LIN {X 0,Y 262.502,Z 609.726,A -85,B 0,C 180,E1 11906.298,E2 11906.298} C_VEL
LIN {X 0,Y 258.219,Z 619.545,A -85,B 0,C 180,E1 11905.702,E2 11905.702} C_VEL
LIN {X 0,Y 254.32,Z 626.854,A -85,B 0,C 180,E1 11904.847,E2 11904.847} C_VEL
LIN {X 0,Y 252.122,Z 630.311,A -85,B 0,C 180,E1 11904.198,E2 11904.198} C_VEL
LIN {X 0,Y 248.406,Z 637.947,A -85,B 0,C 180,E1 11903.61,E2 11903.61} C_VEL
LIN {X 0,Y 245.083,Z 643.553,A -85,B 0,C 180,E1 11902.804,E2 11902.804} C_VEL
LIN {X 0,Y 242.242,Z 647.159,A -85,B 0,C 180,E1 11901.808,E2 11901.808} C_VEL
LIN {X 0,Y 241.54,Z 648.252,A -85,B 0,C 180,E1 11901.619,E2 11901.619} C_VEL
LIN {X 0,Y 238.221,Z 654.054,A -85,B 0,C 180,E1 11900.902,E2 11900.902} C_VEL
LIN {X 0,Y 235.659,Z 657.613,A -85,B 0,C 180,E1 11900.102,E2 11900.102} C_VEL
LIN {X 0,Y 234.291,Z 659.07,A -85,B 0,C 180,E1 11899.444,E2 11899.444} C_VEL
LIN {X 0,Y 233.714,Z 659.362,A -85,B 0,C 180,E1 11898.975,E2 11898.975} C_VEL
LIN {X 0,Y 232.454,Z 676.024,A -85,B 0,C 180,E1 11897.008,E2 11897.008} C_VEL
LIN {X 0,Y 231.033,Z 692.343,A -85,B 0,C 180,E1 11894.538,E2 11894.538} C_VEL
LIN {X 0,Y 229.738,Z 706.728,A -85,B 0,C 180,E1 11891.804,E2 11891.804} C_VEL
LIN {X 0,Y 228.67,Z 719.328,A -85,B 0,C 180,E1 11888.804,E2 11888.804} C_VEL
LIN {X 0,Y 227.959,Z 729.65,A -85,B 0,C 180,E1 11885.791,E2 11885.791} C_VEL
LIN {X 0,Y 227.548,Z 739.398,A -85,B 0,C 180,E1 11882.267,E2 11882.267} C_VEL
LIN {X 0,Y 227.576,Z 746.966,A -85,B 0,C 180,E1 11878.742,E2 11878.742} C_VEL
LIN {X 0,Y 228.06,Z 752.764,A -85,B 0,C 180,E1 11875.223,E2 11875.223} C_VEL
LIN {X 0,Y 229.205,Z 757.315,A -85,B 0,C 180,E1 11871.219,E2 11871.219} C_VEL
LIN {X 0,Y 230.922,Z 759.705,A -85,B 0,C 180,E1 11867.498,E2 11867.498} C_VEL
LIN {X 0,Y 233.318,Z 760.334,A -85,B 0,C 180,E1 11863.827,E2 11863.827} C_VEL
LIN {X 0,Y 236.401,Z 759.155,A -85,B 0,C 180,E1 11860.224,E2 11860.224} C_VEL
LIN {X 0,Y 240.224,Z 756.207,A -85,B 0,C 180,E1 11856.709,E2 11856.709} C_VEL
LIN {X 0,Y 244.74,Z 751.287,A -85,B 0,C 180,E1 11853.296,E2 11853.296} C_VEL
LIN {X 0,Y 249.603,Z 744.876,A -85,B 0,C 180,E1 11850.218,E2 11850.218} C_VEL
LIN {X 0,Y 255.059,Z 736.477,A -85,B 0,C 180,E1 11847.251,E2 11847.251} C_VEL
LIN {X 0,Y 261.105,Z 725.789,A -85,B 0,C 180,E1 11844.405,E2 11844.405} C_VEL
LIN {X 0,Y 263.657,Z 720.912,A -85,B 0,C 180,E1 11843.325,E2 11843.325} C_VEL
LIN {X 0,Y 268.421,Z 719.36,A -85,B 0,C 180,E1 11842.616,E2 11842.616} C_VEL
LIN {X 0,Y 273.025,Z 717.565,A -85,B 0,C 180,E1 11841.999,E2 11841.999} C_VEL
LIN {X 0,Y 266.087,Z 735.239,A -85,B 0,C 180,E1 11839.546,E2 11839.546} C_VEL
LIN {X 0,Y 258.956,Z 751.55,A -85,B 0,C 180,E1 11836.704,E2 11836.704} C_VEL
LIN {X 0,Y 251.798,Z 766.896,A -85,B 0,C 180,E1 11833.39,E2 11833.39} C_VEL
LIN {X 0,Y 245.23,Z 780.336,A -85,B 0,C 180,E1 11829.801,E2 11829.801} C_VEL
LIN {X 0,Y 238.934,Z 792.985,A -85,B 0,C 180,E1 11825.568,E2 11825.568} C_VEL
LIN {X 0,Y 233.562,Z 804.15,A -85,B 0,C 180,E1 11820.911,E2 11820.911} C_VEL
LIN {X 0,Y 229.511,Z 813.251,A -85,B 0,C 180,E1 11816.104,E2 11816.104} C_VEL
LIN {X 0,Y 226.504,Z 821.295,A -85,B 0,C 180,E1 11810.639,E2 11810.639} C_VEL
LIN {X 0,Y 224.934,Z 827.277,A -85,B 0,C 180,E1 11805.204,E2 11805.204} C_VEL
LIN {X 0,Y 224.469,Z 831.288,A -85,B 0,C 180,E1 11800.004,E2 11800.004} C_VEL
LIN {X 0,Y 224.573,Z 833.63,A -85,B 0,C 180,E1 11795.109,E2 11795.109} C_VEL
LIN {X 0,Y 224.701,Z 834.531,A -85,B 0,C 180,E1 11790.765,E2 11790.765} C_VEL
LIN {X 0,Y 224.61,Z 834.309,A -85,B 0,C 180,E1 11786.427,E2 11786.427} C_VEL
LIN {X 0,Y 224.433,Z 832.853,A -85,B 0,C 180,E1 11781.804,E2 11781.804} C_VEL
LIN {X 0,Y 224.637,Z 829.757,A -85,B 0,C 180,E1 11776.617,E2 11776.617} C_VEL
LIN {X 0,Y 225.836,Z 824.839,A -85,B 0,C 180,E1 11771.143,E2 11771.143} C_VEL
LIN {X 0,Y 228.227,Z 818.474,A -85,B 0,C 180,E1 11765.956,E2 11765.956} C_VEL
LIN {X 0,Y 232.239,Z 809.818,A -85,B 0,C 180,E1 11760.606,E2 11760.606} C_VEL
LIN {X 0,Y 237.59,Z 799.573,A -85,B 0,C 180,E1 11755.672,E2 11755.672} C_VEL
LIN {X 0,Y 244.051,Z 787.674,A -85,B 0,C 180,E1 11751.183,E2 11751.183} C_VEL
LIN {X 0,Y 251.363,Z 774.212,A -85,B 0,C 180,E1 11747.14,E2 11747.14} C_VEL
LIN {X 0,Y 259.039,Z 759.532,A -85,B 0,C 180,E1 11743.636,E2 11743.636} C_VEL
LIN {X 0,Y 267.027,Z 743.149,A -85,B 0,C 180,E1 11740.525,E2 11740.525} C_VEL
LIN {X 0,Y 274.424,Z 726.625,A -85,B 0,C 180,E1 11738.005,E2 11738.005} C_VEL
LIN {X 0,Y 281.687,Z 708.409,A -85,B 0,C 180,E1 11735.799,E2 11735.799} C_VEL
LIN {X 0,Y 288.209,Z 689.548,A -85,B 0,C 180,E1 11733.988,E2 11733.988} C_VEL
LIN {X 0,Y 296.028,Z 663.476,A -85,B 0,C 180,E1 11732.029,E2 11732.029} C_VEL
LIN {X 0,Y 299.281,Z 651.866,A -85,B 0,C 180,E1 11731.298,E2 11731.298} C_VEL
LIN {X 0,Y 292.681,Z 660.93,A -85,B 0,C 180,E1 11730.723,E2 11730.723} C_VEL
LIN {X 0,Y 287.143,Z 668.806,A -85,B 0,C 180,E1 11730.324,E2 11730.324} C_VEL
LIN {X 0,Y 282.462,Z 674.515,A -85,B 0,C 180,E1 11729.858,E2 11729.858} C_VEL
LIN {X 0,Y 277.304,Z 680.959,A -85,B 0,C 180,E1 11729.364,E2 11729.364} C_VEL
LIN {X 0,Y 273.388,Z 685.003,A -85,B 0,C 180,E1 11728.865,E2 11728.865} C_VEL
LIN {X 0,Y 268.655,Z 690.182,A -85,B 0,C 180,E1 11728.327,E2 11728.327} C_VEL
LIN {X 0,Y 265.004,Z 693.395,A -85,B 0,C 180,E1 11727.772,E2 11727.772} C_VEL
LIN {X 0,Y 260.584,Z 697.502,A -85,B 0,C 180,E1 11727.167,E2 11727.167} C_VEL
LIN {X 0,Y 258.226,Z 699.12,A -85,B 0,C 180,E1 11726.689,E2 11726.689} C_VEL
LIN {X 0,Y 255.074,Z 711.449,A -85,B 0,C 180,E1 11724.921,E2 11724.921} C_VEL
LIN {X 0,Y 251.112,Z 723.881,A -85,B 0,C 180,E1 11722.595,E2 11722.595} C_VEL
LIN {X 0,Y 247.54,Z 733.199,A -85,B 0,C 180,E1 11720.326,E2 11720.326} C_VEL
LIN {X 0,Y 243.766,Z 741.593,A -85,B 0,C 180,E1 11717.669,E2 11717.669} C_VEL
LIN {X 0,Y 240.065,Z 748.411,A -85,B 0,C 180,E1 11714.717,E2 11714.717} C_VEL
LIN {X 0,Y 236.598,Z 753.609,A -85,B 0,C 180,E1 11711.455,E2 11711.455} C_VEL
LIN {X 0,Y 233.496,Z 756.892,A -85,B 0,C 180,E1 11707.875,E2 11707.875} C_VEL
LIN {X 0,Y 231.206,Z 758.011,A -85,B 0,C 180,E1 11704.464,E2 11704.464} C_VEL
LIN {X 0,Y 229.49,Z 757.302,A -85,B 0,C 180,E1 11700.998,E2 11700.998} C_VEL
LIN {X 0,Y 228.336,Z 754.765,A -85,B 0,C 180,E1 11697.489,E2 11697.489} C_VEL
LIN {X 0,Y 227.7,Z 750.32,A -85,B 0,C 180,E1 11693.95,E2 11693.95} C_VEL
LIN {X 0,Y 227.55,Z 743.766,A -85,B 0,C 180,E1 11690.387,E2 11690.387} C_VEL
LIN {X 0,Y 227.853,Z 735.162,A -85,B 0,C 180,E1 11686.952,E2 11686.952} C_VEL
LIN {X 0,Y 228.469,Z 725.577,A -85,B 0,C 180,E1 11683.995,E2 11683.995} C_VEL
LIN {X 0,Y 229.429,Z 713.354,A -85,B 0,C 180,E1 11681.033,E2 11681.033} C_VEL
LIN {X 0,Y 230.238,Z 703.292,A -85,B 0,C 180,E1 11679.071,E2 11679.071} C_VEL
LIN {X 0,Y 231.431,Z 703.21,A -85,B 0,C 180,E1 11678.188,E2 11678.188} C_VEL
LIN {X 0,Y 234.241,Z 701.447,A -85,B 0,C 180,E1 11677.142,E2 11677.142} C_VEL
LIN {X 0,Y 235.601,Z 700.428,A -85,B 0,C 180,E1 11676.753,E2 11676.753} C_VEL
LIN {X 0,Y 238.132,Z 699.302,A -85,B 0,C 180,E1 11675.663,E2 11675.663} C_VEL
LIN {X 0,Y 242.639,Z 696.175,A -85,B 0,C 180,E1 11674.361,E2 11674.361} C_VEL
LIN {X 0,Y 246.51,Z 693.887,A -85,B 0,C 180,E1 11673.169,E2 11673.169} C_VEL
LIN {X 0,Y 250.791,Z 690.671,A -85,B 0,C 180,E1 11672.194,E2 11672.194} C_VEL
LIN {X 0,Y 255.718,Z 687.371,A -85,B 0,C 180,E1 11670.997,E2 11670.997} C_VEL
LIN {X 0,Y 261.518,Z 682.563,A -85,B 0,C 180,E1 11669.943,E2 11669.943} C_VEL
LIN {X 0,Y 267.1,Z 678.174,A -85,B 0,C 180,E1 11668.895,E2 11668.895} C_VEL
LIN {X 0,Y 273.7,Z 671.73,A -85,B 0,C 180,E1 11668.014,E2 11668.014} C_VEL
LIN {X 0,Y 280.33,Z 665.573,A -85,B 0,C 180,E1 11667.048,E2 11667.048} C_VEL
LIN {X 0,Y 286.573,Z 658.276,A -85,B 0,C 180,E1 11666.425,E2 11666.425} C_VEL
LIN {X 0,Y 289.798,Z 654.217,A -85,B 0,C 180,E1 11666.136,E2 11666.136} C_VEL
LIN {X 0,Y 293.731,Z 649.715,A -85,B 0,C 180,E1 11665.682,E2 11665.682} C_VEL
LIN {X 0,Y 287.854,Z 668.504,A -85,B 0,C 180,E1 11664.031,E2 11664.031} C_VEL
LIN {X 0,Y 281.152,Z 686.562,A -85,B 0,C 180,E1 11662.03,E2 11662.03} C_VEL
LIN {X 0,Y 274.005,Z 703.359,A -85,B 0,C 180,E1 11659.699,E2 11659.699} C_VEL
LIN {X 0,Y 266.569,Z 718.98,A -85,B 0,C 180,E1 11657.006,E2 11657.006} C_VEL
LIN {X 0,Y 259.208,Z 733.136,A -85,B 0,C 180,E1 11653.974,E2 11653.974} C_VEL
LIN {X 0,Y 251.676,Z 746.647,A -85,B 0,C 180,E1 11650.359,E2 11650.359} C_VEL
LIN {X 0,Y 244.708,Z 758.566,A -85,B 0,C 180,E1 11646.332,E2 11646.332} C_VEL
LIN {X 0,Y 238.531,Z 768.9,A -85,B 0,C 180,E1 11641.882,E2 11641.882} C_VEL
LIN {X 0,Y 233.597,Z 777.213,A -85,B 0,C 180,E1 11637.258,E2 11637.258} C_VEL
LIN {X 0,Y 229.734,Z 784.029,A -85,B 0,C 180,E1 11632.25,E2 11632.25} C_VEL
LIN {X 0,Y 227.147,Z 789.026,A -85,B 0,C 180,E1 11627.153,E2 11627.153} C_VEL
LIN {X 0,Y 225.677,Z 792.313,A -85,B 0,C 180,E1 11622.019,E2 11622.019} C_VEL
LIN {X 0,Y 225.034,Z 793.923,A -85,B 0,C 180,E1 11617.147,E2 11617.147} C_VEL
LIN {X 0,Y 224.864,Z 794.129,A -85,B 0,C 180,E1 11612.294,E2 11612.294} C_VEL
LIN {X 0,Y 225.08,Z 792.949,A -85,B 0,C 180,E1 11607.454,E2 11607.454} C_VEL
LIN {X 0,Y 225.864,Z 790.188,A -85,B 0,C 180,E1 11602.368,E2 11602.368} C_VEL
LIN {X 0,Y 227.501,Z 785.806,A -85,B 0,C 180,E1 11597.306,E2 11597.306} C_VEL
LIN {X 0,Y 230.238,Z 779.701,A -85,B 0,C 180,E1 11592.302,E2 11592.302} C_VEL
LIN {X 0,Y 234.194,Z 771.733,A -85,B 0,C 180,E1 11587.403,E2 11587.403} C_VEL
LIN {X 0,Y 239.152,Z 762.251,A -85,B 0,C 180,E1 11582.889,E2 11582.889} C_VEL
LIN {X 0,Y 244.929,Z 751.32,A -85,B 0,C 180,E1 11578.772,E2 11578.772} C_VEL
LIN {X 0,Y 251.343,Z 738.929,A -85,B 0,C 180,E1 11575.035,E2 11575.035} C_VEL
LIN {X 0,Y 258.111,Z 725.195,A -85,B 0,C 180,E1 11571.698,E2 11571.698} C_VEL
LIN {X 0,Y 264.895,Z 710.438,A -85,B 0,C 180,E1 11568.802,E2 11568.802} C_VEL
LIN {X 0,Y 271.694,Z 694.205,A -85,B 0,C 180,E1 11566.222,E2 11566.222} C_VEL
LIN {X 0,Y 278.099,Z 677.046,A -85,B 0,C 180,E1 11564.022,E2 11564.022} C_VEL
LIN {X 0,Y 284.039,Z 658.648,A -85,B 0,C 180,E1 11562.133,E2 11562.133} C_VEL
LIN {X 0,Y 289.114,Z 639.851,A -85,B 0,C 180,E1 11560.614,E2 11560.614} C_VEL
LIN {X 0,Y 293.346,Z 620.178,A -85,B 0,C 180,E1 11559.378,E2 11559.378} C_VEL
LIN {X 0,Y 299.265,Z 586.107,A -85,B 0,C 180,E1 11557.809,E2 11557.809} C_VEL
LIN {X 0,Y 299.981,Z 582.036,A -85,B 0,C 180,E1 11557.649,E2 11557.649} C_VEL
LIN {X 0,Y 300.742,Z 574.657,A -85,B 0,C 180,E1 11557.21,E2 11557.21} C_VEL
LIN {X 0,Y 300.802,Z 555.364,A -85,B 0,C 180,E1 11555.519,E2 11555.519} C_VEL
LIN {X 0,Y 301.467,Z 548.99,A -85,B 0,C 180,E1 11555.181,E2 11555.181} C_VEL
LIN {X 0,Y 307.345,Z 510.718,A -85,B 0,C 180,E1 11553.998,E2 11553.998} C_VEL
LIN {X 0,Y 303.779,Z 519.313,A -85,B 0,C 180,E1 11553.458,E2 11553.458} C_VEL
LIN {X 0,Y 298.05,Z 536.738,A -85,B 0,C 180,E1 11552.901,E2 11552.901} C_VEL
LIN {X 0,Y 292.925,Z 549.446,A -85,B 0,C 180,E1 11552.2,E2 11552.2} C_VEL
LIN {X 0,Y 289.326,Z 557.176,A -85,B 0,C 180,E1 11551.608,E2 11551.608} C_VEL
LIN {X 0,Y 283.915,Z 571.627,A -85,B 0,C 180,E1 11551.031,E2 11551.031} C_VEL
LIN {X 0,Y 278.89,Z 582.682,A -85,B 0,C 180,E1 11550.247,E2 11550.247} C_VEL
LIN {X 0,Y 276.239,Z 587.898,A -85,B 0,C 180,E1 11549.756,E2 11549.756} C_VEL
LIN {X 0,Y 271.205,Z 600.11,A -85,B 0,C 180,E1 11549.167,E2 11549.167} C_VEL
LIN {X 0,Y 266.486,Z 609.396,A -85,B 0,C 180,E1 11548.336,E2 11548.336} C_VEL
LIN {X 0,Y 264.07,Z 613.729,A -85,B 0,C 180,E1 11547.819,E2 11547.819} C_VEL
LIN {X 0,Y 259.544,Z 623.684,A -85,B 0,C 180,E1 11547.197,E2 11547.197} C_VEL
LIN {X 0,Y 255.679,Z 630.673,A -85,B 0,C 180,E1 11546.423,E2 11546.423} C_VEL
LIN {X 0,Y 253.041,Z 634.718,A -85,B 0,C 180,E1 11545.764,E2 11545.764} C_VEL
LIN {X 0,Y 249.16,Z 642.124,A -85,B 0,C 180,E1 11545.175,E2 11545.175} C_VEL
LIN {X 0,Y 245.283,Z 648.292,A -85,B 0,C 180,E1 11544.313,E2 11544.313} C_VEL
LIN {X 0,Y 241.408,Z 653.261,A -85,B 0,C 180,E1 11543.172,E2 11543.172} C_VEL
LIN {X 0,Y 237.624,Z 659.185,A -85,B 0,C 180,E1 11542.384,E2 11542.384} C_VEL
LIN {X 0,Y 234.054,Z 663.75,A -85,B 0,C 180,E1 11541.293,E2 11541.293} C_VEL
LIN {X 0,Y 232.102,Z 665.672,A -85,B 0,C 180,E1 11540.423,E2 11540.423} C_VEL
LIN {X 0,Y 228.336,Z 671.016,A -85,B 0,C 180,E1 11539.44,E2 11539.44} C_VEL
LIN {X 0,Y 226.135,Z 673.635,A -85,B 0,C 180,E1 11538.564,E2 11538.564} C_VEL
LIN {X 0,Y 224.988,Z 674.605,A -85,B 0,C 180,E1 11537.858,E2 11537.858} C_VEL
LIN {X 0,Y 224.681,Z 674.974,A -85,B 0,C 180,E1 11537.525,E2 11537.525} C_VEL
LIN {X 0,Y 223.312,Z 690.47,A -85,B 0,C 180,E1 11535.186,E2 11535.186} C_VEL
LIN {X 0,Y 221.982,Z 704.803,A -85,B 0,C 180,E1 11532.487,E2 11532.487} C_VEL
LIN {X 0,Y 220.824,Z 718.124,A -85,B 0,C 180,E1 11529.382,E2 11529.382} C_VEL
LIN {X 0,Y 219.998,Z 729.809,A -85,B 0,C 180,E1 11526.001,E2 11526.001} C_VEL
LIN {X 0,Y 219.58,Z 739.141,A -85,B 0,C 180,E1 11522.611,E2 11522.611} C_VEL
LIN {X 0,Y 219.585,Z 747.198,A -85,B 0,C 180,E1 11518.957,E2 11518.957} C_VEL
LIN {X 0,Y 220.127,Z 753.726,A -85,B 0,C 180,E1 11515.05,E2 11515.05} C_VEL
LIN {X 0,Y 221.266,Z 758.323,A -85,B 0,C 180,E1 11511.163,E2 11511.163} C_VEL
LIN {X 0,Y 223.083,Z 761.141,A -85,B 0,C 180,E1 11507.314,E2 11507.314} C_VEL
LIN {X 0,Y 225.615,Z 762.137,A -85,B 0,C 180,E1 11503.524,E2 11503.524} C_VEL
LIN {X 0,Y 228.901,Z 761.426,A -85,B 0,C 180,E1 11499.814,E2 11499.814} C_VEL
LIN {X 0,Y 232.951,Z 758.907,A -85,B 0,C 180,E1 11496.206,E2 11496.206} C_VEL
LIN {X 0,Y 237.772,Z 754.592,A -85,B 0,C 180,E1 11492.72,E2 11492.72} C_VEL
LIN {X 0,Y 243.723,Z 747.798,A -85,B 0,C 180,E1 11489.15,E2 11489.15} C_VEL
LIN {X 0,Y 250.039,Z 739.19,A -85,B 0,C 180,E1 11485.957,E2 11485.957} C_VEL
LIN {X 0,Y 256.867,Z 728.653,A -85,B 0,C 180,E1 11483.031,E2 11483.031} C_VEL
LIN {X 0,Y 261.61,Z 727.349,A -85,B 0,C 180,E1 11482.302,E2 11482.302} C_VEL
LIN {X 0,Y 263.699,Z 726.737,A -85,B 0,C 180,E1 11482.003,E2 11482.003} C_VEL
LIN {X 0,Y 256.585,Z 743.146,A -85,B 0,C 180,E1 11479.402,E2 11479.402} C_VEL
LIN {X 0,Y 248.844,Z 759.495,A -85,B 0,C 180,E1 11476.18,E2 11476.18} C_VEL
LIN {X 0,Y 241.751,Z 773.595,A -85,B 0,C 180,E1 11472.71,E2 11472.71} C_VEL
LIN {X 0,Y 234.979,Z 786.571,A -85,B 0,C 180,E1 11468.719,E2 11468.719} C_VEL
LIN {X 0,Y 228.664,Z 798.742,A -85,B 0,C 180,E1 11464.035,E2 11464.035} C_VEL
LIN {X 0,Y 223.722,Z 808.703,A -85,B 0,C 180,E1 11459.153,E2 11459.153} C_VEL
LIN {X 0,Y 219.857,Z 817.56,A -85,B 0,C 180,E1 11453.591,E2 11453.591} C_VEL
LIN {X 0,Y 217.625,Z 824.106,A -85,B 0,C 180,E1 11448.205,E2 11448.205} C_VEL
LIN {X 0,Y 216.604,Z 829.086,A -85,B 0,C 180,E1 11442.53,E2 11442.53} C_VEL
LIN {X 0,Y 216.514,Z 832.069,A -85,B 0,C 180,E1 11437.429,E2 11437.429} C_VEL
LIN {X 0,Y 216.694,Z 833.571,A -85,B 0,C 180,E1 11432.645,E2 11432.645} C_VEL
LIN {X 0,Y 216.709,Z 833.836,A -85,B 0,C 180,E1 11428.414,E2 11428.414} C_VEL
LIN {X 0,Y 216.525,Z 833.028,A -85,B 0,C 180,E1 11423.903,E2 11423.903} C_VEL
LIN {X 0,Y 216.48,Z 830.786,A -85,B 0,C 180,E1 11418.814,E2 11418.814} C_VEL
LIN {X 0,Y 217.242,Z 826.678,A -85,B 0,C 180,E1 11413.144,E2 11413.144} C_VEL
LIN {X 0,Y 219.303,Z 820.827,A -85,B 0,C 180,E1 11407.481,E2 11407.481} C_VEL
LIN {X 0,Y 222.933,Z 813.02,A -85,B 0,C 180,E1 11401.905,E2 11401.905} C_VEL
LIN {X 0,Y 228.256,Z 803.162,A -85,B 0,C 180,E1 11396.5,E2 11396.5} C_VEL
LIN {X 0,Y 234.531,Z 792.163,A -85,B 0,C 180,E1 11391.817,E2 11391.817} C_VEL
LIN {X 0,Y 241.731,Z 779.672,A -85,B 0,C 180,E1 11387.607,E2 11387.607} C_VEL
LIN {X 0,Y 249.571,Z 765.689,A -85,B 0,C 180,E1 11383.851,E2 11383.851} C_VEL
LIN {X 0,Y 257.841,Z 750.026,A -85,B 0,C 180,E1 11380.531,E2 11380.531} C_VEL
LIN {X 0,Y 265.989,Z 733.241,A -85,B 0,C 180,E1 11377.694,E2 11377.694} C_VEL
LIN {X 0,Y 273.506,Z 716.069,A -85,B 0,C 180,E1 11375.39,E2 11375.39} C_VEL
LIN {X 0,Y 280.692,Z 697.229,A -85,B 0,C 180,E1 11373.387,E2 11373.387} C_VEL
LIN {X 0,Y 287.31,Z 677.022,A -85,B 0,C 180,E1 11371.701,E2 11371.701} C_VEL
LIN {X 0,Y 288.035,Z 674.532,A -85,B 0,C 180,E1 11371.495,E2 11371.495} C_VEL
LIN {X 0,Y 284.795,Z 678.348,A -85,B 0,C 180,E1 11371.199,E2 11371.199} C_VEL
LIN {X 0,Y 279.106,Z 685.242,A -85,B 0,C 180,E1 11370.709,E2 11370.709} C_VEL
LIN {X 0,Y 274.44,Z 690.047,A -85,B 0,C 180,E1 11370.183,E2 11370.183} C_VEL
LIN {X 0,Y 269.111,Z 695.424,A -85,B 0,C 180,E1 11369.613,E2 11369.613} C_VEL
LIN {X 0,Y 265.24,Z 698.774,A -85,B 0,C 180,E1 11369.096,E2 11369.096} C_VEL
LIN {X 0,Y 260.319,Z 703.013,A -85,B 0,C 180,E1 11368.441,E2 11368.441} C_VEL
LIN {X 0,Y 257.668,Z 704.9,A -85,B 0,C 180,E1 11368.003,E2 11368.003} C_VEL
LIN {X 0,Y 253.017,Z 708.484,A -85,B 0,C 180,E1 11367.283,E2 11367.283} C_VEL
LIN {X 0,Y 251.309,Z 709.492,A -85,B 0,C 180,E1 11366.908,E2 11366.908} C_VEL
LIN {X 0,Y 247.046,Z 722.372,A -85,B 0,C 180,E1 11364.636,E2 11364.636} C_VEL
LIN {X 0,Y 243.252,Z 731.807,A -85,B 0,C 180,E1 11362.473,E2 11362.473} C_VEL
LIN {X 0,Y 239.028,Z 740.841,A -85,B 0,C 180,E1 11359.804,E2 11359.804} C_VEL
LIN {X 0,Y 234.843,Z 748.248,A -85,B 0,C 180,E1 11356.828,E2 11356.828} C_VEL
LIN {X 0,Y 231.134,Z 753.659,A -85,B 0,C 180,E1 11353.763,E2 11353.763} C_VEL
LIN {X 0,Y 227.471,Z 757.673,A -85,B 0,C 180,E1 11350.126,E2 11350.126} C_VEL
LIN {X 0,Y 224.682,Z 759.426,A -85,B 0,C 180,E1 11346.643,E2 11346.643} C_VEL
LIN {X 0,Y 222.525,Z 759.381,A -85,B 0,C 180,E1 11343.09,E2 11343.09} C_VEL
LIN {X 0,Y 220.981,Z 757.506,A -85,B 0,C 180,E1 11339.467,E2 11339.467} C_VEL
LIN {X 0,Y 220.02,Z 753.773,A -85,B 0,C 180,E1 11335.829,E2 11335.829} C_VEL
LIN {X 0,Y 219.594,Z 748.018,A -85,B 0,C 180,E1 11332.148,E2 11332.148} C_VEL
LIN {X 0,Y 219.659,Z 740.652,A -85,B 0,C 180,E1 11328.712,E2 11328.712} C_VEL
LIN {X 0,Y 220.055,Z 732.621,A -85,B 0,C 180,E1 11325.796,E2 11325.796} C_VEL
LIN {X 0,Y 220.784,Z 722.414,A -85,B 0,C 180,E1 11322.854,E2 11322.854} C_VEL
LIN {X 0,Y 221.632,Z 712.076,A -85,B 0,C 180,E1 11320.428,E2 11320.428} C_VEL
LIN {X 0,Y 222.704,Z 712.025,A -85,B 0,C 180,E1 11319.5,E2 11319.5} C_VEL
LIN {X 0,Y 225.293,Z 710.531,A -85,B 0,C 180,E1 11318.385,E2 11318.385} C_VEL
LIN {X 0,Y 226.512,Z 709.719,A -85,B 0,C 180,E1 11317.962,E2 11317.962} C_VEL
LIN {X 0,Y 229.325,Z 708.521,A -85,B 0,C 180,E1 11316.623,E2 11316.623} C_VEL
LIN {X 0,Y 232.499,Z 706.475,A -85,B 0,C 180,E1 11315.615,E2 11315.615} C_VEL
LIN {X 0,Y 236.428,Z 704.454,A -85,B 0,C 180,E1 11314.176,E2 11314.176} C_VEL
LIN {X 0,Y 239.929,Z 702.116,A -85,B 0,C 180,E1 11313.251,E2 11313.251} C_VEL
LIN {X 0,Y 245.082,Z 699.143,A -85,B 0,C 180,E1 11311.79,E2 11311.79} C_VEL
LIN {X 0,Y 249.07,Z 696.322,A -85,B 0,C 180,E1 11310.938,E2 11310.938} C_VEL
LIN {X 0,Y 254.197,Z 693.037,A -85,B 0,C 180,E1 11309.769,E2 11309.769} C_VEL
LIN {X 0,Y 261.559,Z 687.358,A -85,B 0,C 180,E1 11308.481,E2 11308.481} C_VEL
LIN {X 0,Y 268.267,Z 682.136,A -85,B 0,C 180,E1 11307.387,E2 11307.387} C_VEL
LIN {X 0,Y 274.442,Z 676.361,A -85,B 0,C 180,E1 11306.623,E2 11306.623} C_VEL
LIN {X 0,Y 281.874,Z 669.607,A -85,B 0,C 180,E1 11305.666,E2 11305.666} C_VEL
LIN {X 0,Y 283.658,Z 667.723,A -85,B 0,C 180,E1 11305.484,E2 11305.484} C_VEL
LIN {X 0,Y 276.77,Z 685.962,A -85,B 0,C 180,E1 11303.491,E2 11303.491} C_VEL
LIN {X 0,Y 269.199,Z 703.305,A -85,B 0,C 180,E1 11301.118,E2 11301.118} C_VEL
LIN {X 0,Y 261.356,Z 719.201,A -85,B 0,C 180,E1 11298.387,E2 11298.387} C_VEL
LIN {X 0,Y 253.443,Z 733.798,A -85,B 0,C 180,E1 11295.245,E2 11295.245} C_VEL
LIN {X 0,Y 245.541,Z 747.305,A -85,B 0,C 180,E1 11291.587,E2 11291.587} C_VEL
LIN {X 0,Y 238.198,Z 759.215,A -85,B 0,C 180,E1 11287.493,E2 11287.493} C_VEL
LIN {X 0,Y 231.962,Z 769.057,A -85,B 0,C 180,E1 11283.191,E2 11283.191} C_VEL
LIN {X 0,Y 226.627,Z 777.477,A -85,B 0,C 180,E1 11278.457,E2 11278.457} C_VEL
LIN {X 0,Y 222.404,Z 784.395,A -85,B 0,C 180,E1 11273.305,E2 11273.305} C_VEL
LIN {X 0,Y 219.527,Z 789.487,A -85,B 0,C 180,E1 11268.042,E2 11268.042} C_VEL
LIN {X 0,Y 217.858,Z 792.865,A -85,B 0,C 180,E1 11262.727,E2 11262.727} C_VEL
LIN {X 0,Y 217.113,Z 794.569,A -85,B 0,C 180,E1 11257.675,E2 11257.675} C_VEL
LIN {X 0,Y 216.895,Z 794.873,A -85,B 0,C 180,E1 11252.642,E2 11252.642} C_VEL
LIN {X 0,Y 217.098,Z 793.795,A -85,B 0,C 180,E1 11247.624,E2 11247.624} C_VEL
LIN {X 0,Y 217.893,Z 791.169,A -85,B 0,C 180,E1 11242.389,E2 11242.389} C_VEL
LIN {X 0,Y 219.602,Z 786.875,A -85,B 0,C 180,E1 11237.109,E2 11237.109} C_VEL
LIN {X 0,Y 222.457,Z 780.888,A -85,B 0,C 180,E1 11231.933,E2 11231.933} C_VEL
LIN {X 0,Y 226.589,Z 773.048,A -85,B 0,C 180,E1 11226.876,E2 11226.876} C_VEL
LIN {X 0,Y 231.762,Z 763.711,A -85,B 0,C 180,E1 11222.229,E2 11222.229} C_VEL
LIN {X 0,Y 238.143,Z 752.289,A -85,B 0,C 180,E1 11217.777,E2 11217.777} C_VEL
LIN {X 0,Y 244.931,Z 739.808,A -85,B 0,C 180,E1 11213.93,E2 11213.93} C_VEL
LIN {X 0,Y 251.922,Z 726.251,A -85,B 0,C 180,E1 11210.578,E2 11210.578} C_VEL
LIN {X 0,Y 258.983,Z 711.57,A -85,B 0,C 180,E1 11207.647,E2 11207.647} C_VEL
LIN {X 0,Y 266.041,Z 695.428,A -85,B 0,C 180,E1 11205.044,E2 11205.044} C_VEL
LIN {X 0,Y 272.959,Z 677.597,A -85,B 0,C 180,E1 11202.74,E2 11202.74} C_VEL
LIN {X 0,Y 279.008,Z 659.414,A -85,B 0,C 180,E1 11200.874,E2 11200.874} C_VEL
LIN {X 0,Y 284.355,Z 640.233,A -85,B 0,C 180,E1 11199.324,E2 11199.324} C_VEL
LIN {X 0,Y 288.711,Z 620.576,A -85,B 0,C 180,E1 11198.093,E2 11198.093} C_VEL
LIN {X 0,Y 294.87,Z 586.485,A -85,B 0,C 180,E1 11196.521,E2 11196.521} C_VEL
LIN {X 0,Y 301.467,Z 548.99,A -85,B 0,C 180,E1 11195.181,E2 11195.181} C_VEL
LIN {X 0,Y 300.991,Z 548.293,A -85,B 0,C 180,E1 11194.96,E2 11194.96} C_VEL
LIN {X 0,Y 299.609,Z 549.011,A -85,B 0,C 180,E1 11194.562,E2 11194.562} C_VEL
LIN {X 0,Y 297.222,Z 551.853,A -85,B 0,C 180,E1 11194.006,E2 11194.006} C_VEL
LIN {X 0,Y 292.455,Z 560.378,A -85,B 0,C 180,E1 11193.12,E2 11193.12} C_VEL
LIN {X 0,Y 289.967,Z 566.074,A -85,B 0,C 180,E1 11192.793,E2 11192.793} C_VEL
LIN {X 0,Y 284.271,Z 579.799,A -85,B 0,C 180,E1 11192.126,E2 11192.126} C_VEL
LIN {X 0,Y 279.182,Z 589.921,A -85,B 0,C 180,E1 11191.286,E2 11191.286} C_VEL
LIN {X 0,Y 272.828,Z 604.656,A -85,B 0,C 180,E1 11190.545,E2 11190.545} C_VEL
LIN {X 0,Y 267.692,Z 614.365,A -85,B 0,C 180,E1 11189.664,E2 11189.664} C_VEL
LIN {X 0,Y 265.81,Z 617.679,A -85,B 0,C 180,E1 11189.318,E2 11189.318} C_VEL
LIN {X 0,Y 260.96,Z 627.92,A -85,B 0,C 180,E1 11188.668,E2 11188.668} C_VEL
LIN {X 0,Y 256.305,Z 635.851,A -85,B 0,C 180,E1 11187.787,E2 11187.787} C_VEL
LIN {X 0,Y 254.048,Z 639.206,A -85,B 0,C 180,E1 11187.305,E2 11187.305} C_VEL
LIN {X 0,Y 249.385,Z 647.408,A -85,B 0,C 180,E1 11186.61,E2 11186.61} C_VEL
LIN {X 0,Y 244.787,Z 653.885,A -85,B 0,C 180,E1 11185.657,E2 11185.657} C_VEL
LIN {X 0,Y 241.404,Z 658.108,A -85,B 0,C 180,E1 11184.73,E2 11184.73} C_VEL
LIN {X 0,Y 236.67,Z 664.698,A -85,B 0,C 180,E1 11183.796,E2 11183.796} C_VEL
LIN {X 0,Y 232.993,Z 669.168,A -85,B 0,C 180,E1 11182.721,E2 11182.721} C_VEL
LIN {X 0,Y 230.504,Z 671.728,A -85,B 0,C 180,E1 11181.832,E2 11181.832} C_VEL
LIN {X 0,Y 226.232,Z 677.064,A -85,B 0,C 180,E1 11180.707,E2 11180.707} C_VEL
LIN {X 0,Y 223.486,Z 679.982,A -85,B 0,C 180,E1 11179.607,E2 11179.607} C_VEL
LIN {X 0,Y 222.171,Z 681.174,A -85,B 0,C 180,E1 11178.908,E2 11178.908} C_VEL
LIN {X 0,Y 218.745,Z 685.321,A -85,B 0,C 180,E1 11177.834,E2 11177.834} C_VEL
LIN {X 0,Y 216.399,Z 687.719,A -85,B 0,C 180,E1 11176.648,E2 11176.648} C_VEL
LIN {X 0,Y 215.612,Z 688.29,A -85,B 0,C 180,E1 11175.88,E2 11175.88} C_VEL
LIN {X 0,Y 214.136,Z 703.999,A -85,B 0,C 180,E1 11172.952,E2 11172.952} C_VEL
LIN {X 0,Y 212.91,Z 717.749,A -85,B 0,C 180,E1 11169.734,E2 11169.734} C_VEL
LIN {X 0,Y 212.082,Z 728.893,A -85,B 0,C 180,E1 11166.498,E2 11166.498} C_VEL
LIN {X 0,Y 211.616,Z 738.799,A -85,B 0,C 180,E1 11162.98,E2 11162.98} C_VEL
LIN {X 0,Y 211.586,Z 747.258,A -85,B 0,C 180,E1 11159.189,E2 11159.189} C_VEL
LIN {X 0,Y 212.076,Z 753.845,A -85,B 0,C 180,E1 11155.404,E2 11155.404} C_VEL
LIN {X 0,Y 213.318,Z 759.257,A -85,B 0,C 180,E1 11151.103,E2 11151.103} C_VEL
LIN {X 0,Y 215.222,Z 762.439,A -85,B 0,C 180,E1 11147.116,E2 11147.116} C_VEL
LIN {X 0,Y 217.911,Z 763.907,A -85,B 0,C 180,E1 11143.199,E2 11143.199} C_VEL
LIN {X 0,Y 221.387,Z 763.597,A -85,B 0,C 180,E1 11139.374,E2 11139.374} C_VEL
LIN {X 0,Y 226.015,Z 761.415,A -85,B 0,C 180,E1 11135.429,E2 11135.429} C_VEL
LIN {X 0,Y 231.54,Z 757.16,A -85,B 0,C 180,E1 11131.641,E2 11131.641} C_VEL
LIN {X 0,Y 237.529,Z 751.244,A -85,B 0,C 180,E1 11128.253,E2 11128.253} C_VEL
LIN {X 0,Y 243.805,Z 743.925,A -85,B 0,C 180,E1 11125.247,E2 11125.247} C_VEL
LIN {X 0,Y 249.841,Z 735.968,A -85,B 0,C 180,E1 11122.75,E2 11122.75} C_VEL
LIN {X 0,Y 254.348,Z 734.969,A -85,B 0,C 180,E1 11121.998,E2 11121.998} C_VEL
LIN {X 0,Y 246.683,Z 751.137,A -85,B 0,C 180,E1 11119.107,E2 11119.107} C_VEL
LIN {X 0,Y 239.37,Z 765.476,A -85,B 0,C 180,E1 11115.927,E2 11115.927} C_VEL
LIN {X 0,Y 232.095,Z 778.95,A -85,B 0,C 180,E1 11112.187,E2 11112.187} C_VEL
LIN {X 0,Y 225.029,Z 791.753,A -85,B 0,C 180,E1 11107.732,E2 11107.732} C_VEL
LIN {X 0,Y 219.05,Z 802.809,A -85,B 0,C 180,E1 11102.875,E2 11102.875} C_VEL
LIN {X 0,Y 214.248,Z 812.279,A -85,B 0,C 180,E1 11097.517,E2 11097.517} C_VEL
LIN {X 0,Y 210.863,Z 820.217,A -85,B 0,C 180,E1 11091.707,E2 11091.707} C_VEL
LIN {X 0,Y 209.084,Z 825.966,A -85,B 0,C 180,E1 11086.016,E2 11086.016} C_VEL
LIN {X 0,Y 208.51,Z 830.066,A -85,B 0,C 180,E1 11080.22,E2 11080.22} C_VEL
LIN {X 0,Y 208.623,Z 832.24,A -85,B 0,C 180,E1 11075.225,E2 11075.225} C_VEL
LIN {X 0,Y 208.767,Z 833.108,A -85,B 0,C 180,E1 11070.549,E2 11070.549} C_VEL
LIN {X 0,Y 208.645,Z 832.834,A -85,B 0,C 180,E1 11065.878,E2 11065.878} C_VEL
LIN {X 0,Y 208.458,Z 831.307,A -85,B 0,C 180,E1 11060.893,E2 11060.893} C_VEL
LIN {X 0,Y 208.82,Z 828.118,A -85,B 0,C 180,E1 11055.282,E2 11055.282} C_VEL
LIN {X 0,Y 210.392,Z 823.107,A -85,B 0,C 180,E1 11049.41,E2 11049.41} C_VEL
LIN {X 0,Y 213.527,Z 816.237,A -85,B 0,C 180,E1 11043.586,E2 11043.586} C_VEL
LIN {X 0,Y 218.463,Z 807.248,A -85,B 0,C 180,E1 11037.854,E2 11037.854} C_VEL
LIN {X 0,Y 224.672,Z 796.865,A -85,B 0,C 180,E1 11032.753,E2 11032.753} C_VEL
LIN {X 0,Y 232.08,Z 784.682,A -85,B 0,C 180,E1 11028.103,E2 11028.103} C_VEL
LIN {X 0,Y 240.206,Z 771.163,A -85,B 0,C 180,E1 11024.037,E2 11024.037} C_VEL
LIN {X 0,Y 248.618,Z 756.355,A -85,B 0,C 180,E1 11020.527,E2 11020.527} C_VEL
LIN {X 0,Y 257.111,Z 740.223,A -85,B 0,C 180,E1 11017.503,E2 11017.503} C_VEL
LIN {X 0,Y 265.351,Z 723.019,A -85,B 0,C 180,E1 11014.941,E2 11014.941} C_VEL
LIN {X 0,Y 272.895,Z 705.104,A -85,B 0,C 180,E1 11012.837,E2 11012.837} C_VEL
LIN {X 0,Y 277.309,Z 693.094,A -85,B 0,C 180,E1 11011.645,E2 11011.645} C_VEL
LIN {X 0,Y 270.115,Z 700.183,A -85,B 0,C 180,E1 11010.965,E2 11010.965} C_VEL
LIN {X 0,Y 264.514,Z 704.956,A -85,B 0,C 180,E1 11010.306,E2 11010.306} C_VEL
LIN {X 0,Y 258.402,Z 709.543,A -85,B 0,C 180,E1 11009.469,E2 11009.469} C_VEL
LIN {X 0,Y 252.487,Z 713.852,A -85,B 0,C 180,E1 11008.63,E2 11008.63} C_VEL
LIN {X 0,Y 248.905,Z 716.175,A -85,B 0,C 180,E1 11008.033,E2 11008.033} C_VEL
LIN {X 0,Y 244.19,Z 719.001,A -85,B 0,C 180,E1 11007.098,E2 11007.098} C_VEL
LIN {X 0,Y 239.861,Z 729.564,A -85,B 0,C 180,E1 11004.898,E2 11004.898} C_VEL
LIN {X 0,Y 235.12,Z 739.395,A -85,B 0,C 180,E1 11002.238,E2 11002.238} C_VEL
LIN {X 0,Y 230.38,Z 747.537,A -85,B 0,C 180,E1 10999.258,E2 10999.258} C_VEL
LIN {X 0,Y 226.117,Z 753.563,A -85,B 0,C 180,E1 10996.174,E2 10996.174} C_VEL
LIN {X 0,Y 222.108,Z 758.028,A -85,B 0,C 180,E1 10992.742,E2 10992.742} C_VEL
LIN {X 0,Y 218.729,Z 760.534,A -85,B 0,C 180,E1 10989.206,E2 10989.206} C_VEL
LIN {X 0,Y 216.029,Z 761.261,A -85,B 0,C 180,E1 10985.577,E2 10985.577} C_VEL
LIN {X 0,Y 213.868,Z 760.015,A -85,B 0,C 180,E1 10981.606,E2 10981.606} C_VEL
LIN {X 0,Y 212.449,Z 756.65,A -85,B 0,C 180,E1 10977.571,E2 10977.571} C_VEL
LIN {X 0,Y 211.748,Z 751.515,A -85,B 0,C 180,E1 10973.764,E2 10973.764} C_VEL
LIN {X 0,Y 211.598,Z 744.789,A -85,B 0,C 180,E1 10970.205,E2 10970.205} C_VEL
LIN {X 0,Y 211.875,Z 736.656,A -85,B 0,C 180,E1 10966.907,E2 10966.907} C_VEL
LIN {X 0,Y 212.532,Z 726.544,A -85,B 0,C 180,E1 10963.684,E2 10963.684} C_VEL
LIN {X 0,Y 213.056,Z 720.295,A -85,B 0,C 180,E1 10961.956,E2 10961.956} C_VEL
LIN {X 0,Y 214.143,Z 720.167,A -85,B 0,C 180,E1 10960.922,E2 10960.922} C_VEL
LIN {X 0,Y 216.577,Z 718.812,A -85,B 0,C 180,E1 10959.741,E2 10959.741} C_VEL
LIN {X 0,Y 217.549,Z 718.301,A -85,B 0,C 180,E1 10959.273,E2 10959.273} C_VEL
LIN {X 0,Y 220.27,Z 717.176,A -85,B 0,C 180,E1 10957.822,E2 10957.822} C_VEL
LIN {X 0,Y 223.036,Z 715.603,A -85,B 0,C 180,E1 10956.764,E2 10956.764} C_VEL
LIN {X 0,Y 226.924,Z 713.756,A -85,B 0,C 180,E1 10955.186,E2 10955.186} C_VEL
LIN {X 0,Y 229.717,Z 712.129,A -85,B 0,C 180,E1 10954.289,E2 10954.289} C_VEL
LIN {X 0,Y 234.218,Z 709.791,A -85,B 0,C 180,E1 10952.82,E2 10952.82} C_VEL
LIN {X 0,Y 237.784,Z 707.635,A -85,B 0,C 180,E1 10951.903,E2 10951.903} C_VEL
LIN {X 0,Y 243.34,Z 704.501,A -85,B 0,C 180,E1 10950.457,E2 10950.457} C_VEL
LIN {X 0,Y 248.046,Z 701.431,A -85,B 0,C 180,E1 10949.475,E2 10949.475} C_VEL
LIN {X 0,Y 254.309,Z 697.407,A -85,B 0,C 180,E1 10948.207,E2 10948.207} C_VEL
LIN {X 0,Y 260.464,Z 692.859,A -85,B 0,C 180,E1 10947.229,E2 10947.229} C_VEL
LIN {X 0,Y 267.42,Z 687.726,A -85,B 0,C 180,E1 10946.144,E2 10946.144} C_VEL
LIN {X 0,Y 273.998,Z 681.906,A -85,B 0,C 180,E1 10945.407,E2 10945.407} C_VEL
LIN {X 0,Y 266.247,Z 699.598,A -85,B 0,C 180,E1 10943.121,E2 10943.121} C_VEL
LIN {X 0,Y 258.07,Z 716.044,A -85,B 0,C 180,E1 10940.445,E2 10940.445} C_VEL
LIN {X 0,Y 249.872,Z 730.879,A -85,B 0,C 180,E1 10937.416,E2 10937.416} C_VEL
LIN {X 0,Y 241.872,Z 744.245,A -85,B 0,C 180,E1 10933.987,E2 10933.987} C_VEL
LIN {X 0,Y 234.255,Z 756.18,A -85,B 0,C 180,E1 10930.129,E2 10930.129} C_VEL
LIN {X 0,Y 227.265,Z 766.691,A -85,B 0,C 180,E1 10925.813,E2 10925.813} C_VEL
LIN {X 0,Y 221.162,Z 775.734,A -85,B 0,C 180,E1 10921.024,E2 10921.024} C_VEL
LIN {X 0,Y 216.169,Z 783.217,A -85,B 0,C 180,E1 10915.772,E2 10915.772} C_VEL
LIN {X 0,Y 212.626,Z 788.839,A -85,B 0,C 180,E1 10910.364,E2 10910.364} C_VEL
LIN {X 0,Y 210.432,Z 792.732,A -85,B 0,C 180,E1 10904.867,E2 10904.867} C_VEL
LIN {X 0,Y 209.324,Z 794.991,A -85,B 0,C 180,E1 10899.347,E2 10899.347} C_VEL
LIN {X 0,Y 208.952,Z 795.689,A -85,B 0,C 180,E1 10894.116,E2 10894.116} C_VEL
LIN {X 0,Y 209.043,Z 794.961,A -85,B 0,C 180,E1 10888.904,E2 10888.904} C_VEL
LIN {X 0,Y 209.651,Z 792.854,A -85,B 0,C 180,E1 10883.703,E2 10883.703} C_VEL
LIN {X 0,Y 211.15,Z 789.104,A -85,B 0,C 180,E1 10878.251,E2 10878.251} C_VEL
LIN {X 0,Y 213.813,Z 783.68,A -85,B 0,C 180,E1 10872.866,E2 10872.866} C_VEL
LIN {X 0,Y 217.796,Z 776.467,A -85,B 0,C 180,E1 10867.602,E2 10867.602} C_VEL
LIN {X 0,Y 222.865,Z 767.787,A -85,B 0,C 180,E1 10862.767,E2 10862.767} C_VEL
LIN {X 0,Y 228.82,Z 757.713,A -85,B 0,C 180,E1 10858.375,E2 10858.375} C_VEL
LIN {X 0,Y 235.866,Z 745.607,A -85,B 0,C 180,E1 10854.197,E2 10854.197} C_VEL
LIN {X 0,Y 243.455,Z 731.902,A -85,B 0,C 180,E1 10850.463,E2 10850.463} C_VEL
LIN {X 0,Y 251.098,Z 716.994,A -85,B 0,C 180,E1 10847.24,E2 10847.24} C_VEL
LIN {X 0,Y 258.562,Z 701.061,A -85,B 0,C 180,E1 10844.482,E2 10844.482} C_VEL
LIN {X 0,Y 265.622,Z 684.145,A -85,B 0,C 180,E1 10842.136,E2 10842.136} C_VEL
LIN {X 0,Y 272.406,Z 665.402,A -85,B 0,C 180,E1 10840.066,E2 10840.066} C_VEL
LIN {X 0,Y 277.952,Z 647.286,A -85,B 0,C 180,E1 10838.487,E2 10838.487} C_VEL
LIN {X 0,Y 282.739,Z 628.08,A -85,B 0,C 180,E1 10837.168,E2 10837.168} C_VEL
LIN {X 0,Y 287.664,Z 602.819,A -85,B 0,C 180,E1 10835.875,E2 10835.875} C_VEL
LIN {X 0,Y 295.043,Z 563.107,A -85,B 0,C 180,E1 10834.317,E2 10834.317} C_VEL
LIN {X 0,Y 297.637,Z 548.184,A -85,B 0,C 180,E1 10833.803,E2 10833.803} C_VEL
LIN {X 0,Y 292.036,Z 560.418,A -85,B 0,C 180,E1 10832.97,E2 10832.97} C_VEL
LIN {X 0,Y 289.967,Z 566.074,A -85,B 0,C 180,E1 10832.793,E2 10832.793} C_VEL
LIN {X 0,Y 286.529,Z 576.558,A -85,B 0,C 180,E1 10832.616,E2 10832.616} C_VEL
LIN {X 0,Y 281.001,Z 594.573,A -85,B 0,C 180,E1 10832.572,E2 10832.572} C_VEL
LIN {X 0,Y 278.995,Z 599.669,A -85,B 0,C 180,E1 10832.426,E2 10832.426} C_VEL
LIN {X 0,Y 273.482,Z 611.407,A -85,B 0,C 180,E1 10831.737,E2 10831.737} C_VEL
LIN {X 0,Y 267.766,Z 621.662,A -85,B 0,C 180,E1 10830.785,E2 10830.785} C_VEL
LIN {X 0,Y 262.36,Z 632.368,A -85,B 0,C 180,E1 10830.105,E2 10830.105} C_VEL
LIN {X 0,Y 257.119,Z 640.604,A -85,B 0,C 180,E1 10829.212,E2 10829.212} C_VEL
LIN {X 0,Y 255.06,Z 643.731,A -85,B 0,C 180,E1 10828.828,E2 10828.828} C_VEL
LIN {X 0,Y 249.655,Z 652.403,A -85,B 0,C 180,E1 10828.073,E2 10828.073} C_VEL
LIN {X 0,Y 245.013,Z 658.588,A -85,B 0,C 180,E1 10827.173,E2 10827.173} C_VEL
LIN {X 0,Y 241.422,Z 662.764,A -85,B 0,C 180,E1 10826.306,E2 10826.306} C_VEL
LIN {X 0,Y 236.183,Z 669.653,A -85,B 0,C 180,E1 10825.315,E2 10825.315} C_VEL
LIN {X 0,Y 231.874,Z 674.445,A -85,B 0,C 180,E1 10824.184,E2 10824.184} C_VEL
LIN {X 0,Y 229.017,Z 677.429,A -85,B 0,C 180,E1 10823.274,E2 10823.274} C_VEL
LIN {X 0,Y 224.142,Z 682.924,A -85,B 0,C 180,E1 10822.007,E2 10822.007} C_VEL
LIN {X 0,Y 220.724,Z 686.201,A -85,B 0,C 180,E1 10820.692,E2 10820.692} C_VEL
LIN {X 0,Y 219.485,Z 687.442,A -85,B 0,C 180,E1 10820.209,E2 10820.209} C_VEL
LIN {X 0,Y 215.607,Z 691.673,A -85,B 0,C 180,E1 10818.908,E2 10818.908} C_VEL
LIN {X 0,Y 212.859,Z 694.15,A -85,B 0,C 180,E1 10817.496,E2 10817.496} C_VEL
LIN {X 0,Y 212.24,Z 694.685,A -85,B 0,C 180,E1 10817.125,E2 10817.125} C_VEL
LIN {X 0,Y 208.831,Z 698.474,A -85,B 0,C 180,E1 10815.768,E2 10815.768} C_VEL
LIN {X 0,Y 206.994,Z 700.19,A -85,B 0,C 180,E1 10814.548,E2 10814.548} C_VEL
LIN {X 0,Y 206.529,Z 700.604,A -85,B 0,C 180,E1 10813.938,E2 10813.938} C_VEL
LIN {X 0,Y 205.141,Z 715.545,A -85,B 0,C 180,E1 10810.533,E2 10810.533} C_VEL
LIN {X 0,Y 204.123,Z 728.752,A -85,B 0,C 180,E1 10806.752,E2 10806.752} C_VEL
LIN {X 0,Y 203.628,Z 738.935,A -85,B 0,C 180,E1 10803.097,E2 10803.097} C_VEL
LIN {X 0,Y 203.6,Z 747.747,A -85,B 0,C 180,E1 10799.157,E2 10799.157} C_VEL
LIN {X 0,Y 204.186,Z 755.044,A -85,B 0,C 180,E1 10794.944,E2 10794.944} C_VEL
LIN {X 0,Y 205.46,Z 760.327,A -85,B 0,C 180,E1 10790.76,E2 10790.76} C_VEL
LIN {X 0,Y 207.518,Z 763.871,A -85,B 0,C 180,E1 10786.629,E2 10786.629} C_VEL
LIN {X 0,Y 210.63,Z 765.67,A -85,B 0,C 180,E1 10782.315,E2 10782.315} C_VEL
LIN {X 0,Y 214.437,Z 765.627,A -85,B 0,C 180,E1 10778.387,E2 10778.387} C_VEL
LIN {X 0,Y 219.805,Z 763.531,A -85,B 0,C 180,E1 10774.108,E2 10774.108} C_VEL
LIN {X 0,Y 225.83,Z 759.492,A -85,B 0,C 180,E1 10770.273,E2 10770.273} C_VEL
LIN {X 0,Y 232.33,Z 753.89,A -85,B 0,C 180,E1 10766.87,E2 10766.87} C_VEL
LIN {X 0,Y 239.865,Z 746.102,A -85,B 0,C 180,E1 10763.563,E2 10763.563} C_VEL
LIN {X 0,Y 242.745,Z 742.797,A -85,B 0,C 180,E1 10762.44,E2 10762.44} C_VEL
LIN {X 0,Y 244.93,Z 742.628,A -85,B 0,C 180,E1 10761.987,E2 10761.987} C_VEL
LIN {X 0,Y 236.807,Z 758.413,A -85,B 0,C 180,E1 10758.802,E2 10758.802} C_VEL
LIN {X 0,Y 228.733,Z 772.939,A -85,B 0,C 180,E1 10755.085,E2 10755.085} C_VEL
LIN {X 0,Y 221.294,Z 785.861,A -85,B 0,C 180,E1 10750.931,E2 10750.931} C_VEL
LIN {X 0,Y 214.629,Z 797.344,A -85,B 0,C 180,E1 10746.273,E2 10746.273} C_VEL
LIN {X 0,Y 209.019,Z 807.31,A -85,B 0,C 180,E1 10741.102,E2 10741.102} C_VEL
LIN {X 0,Y 204.673,Z 815.956,A -85,B 0,C 180,E1 10735.346,E2 10735.346} C_VEL
LIN {X 0,Y 202.038,Z 822.45,A -85,B 0,C 180,E1 10729.665,E2 10729.665} C_VEL
LIN {X 0,Y 200.719,Z 827.509,A -85,B 0,C 180,E1 10723.54,E2 10723.54} C_VEL
LIN {X 0,Y 200.541,Z 830.559,A -85,B 0,C 180,E1 10718.025,E2 10718.025} C_VEL
LIN {X 0,Y 200.735,Z 832.063,A -85,B 0,C 180,E1 10713.141,E2 10713.141} C_VEL
LIN {X 0,Y 200.775,Z 832.43,A -85,B 0,C 180,E1 10708.573,E2 10708.573} C_VEL
LIN {X 0,Y 200.569,Z 831.702,A -85,B 0,C 180,E1 10703.703,E2 10703.703} C_VEL
LIN {X 0,Y 200.536,Z 829.525,A -85,B 0,C 180,E1 10698.204,E2 10698.204} C_VEL
LIN {X 0,Y 201.484,Z 825.464,A -85,B 0,C 180,E1 10692.081,E2 10692.081} C_VEL
LIN {X 0,Y 203.932,Z 819.661,A -85,B 0,C 180,E1 10685.987,E2 10685.987} C_VEL
LIN {X 0,Y 207.886,Z 812.372,A -85,B 0,C 180,E1 10680.304,E2 10680.304} C_VEL
LIN {X 0,Y 213.518,Z 803.154,A -85,B 0,C 180,E1 10674.831,E2 10674.831} C_VEL
LIN {X 0,Y 220.798,Z 791.864,A -85,B 0,C 180,E1 10669.642,E2 10669.642} C_VEL
LIN {X 0,Y 228.696,Z 779.57,A -85,B 0,C 180,E1 10665.259,E2 10665.259} C_VEL
LIN {X 0,Y 237.231,Z 765.765,A -85,B 0,C 180,E1 10661.39,E2 10661.39} C_VEL
LIN {X 0,Y 246.173,Z 750.442,A -85,B 0,C 180,E1 10658.005,E2 10658.005} C_VEL
LIN {X 0,Y 254.918,Z 733.944,A -85,B 0,C 180,E1 10655.135,E2 10655.135} C_VEL
LIN {X 0,Y 263.155,Z 716.684,A -85,B 0,C 180,E1 10652.765,E2 10652.765} C_VEL
LIN {X 0,Y 266.588,Z 708.615,A -85,B 0,C 180,E1 10651.812,E2 10651.812} C_VEL
LIN {X 0,Y 259.821,Z 713.806,A -85,B 0,C 180,E1 10651.041,E2 10651.041} C_VEL
LIN {X 0,Y 251.114,Z 719.655,A -85,B 0,C 180,E1 10649.848,E2 10649.848} C_VEL
LIN {X 0,Y 243.86,Z 723.928,A -85,B 0,C 180,E1 10648.666,E2 10648.666} C_VEL
LIN {X 0,Y 237.852,Z 727.092,A -85,B 0,C 180,E1 10647.542,E2 10647.542} C_VEL
LIN {X 0,Y 236.839,Z 727.765,A -85,B 0,C 180,E1 10647.261,E2 10647.261} C_VEL
LIN {X 0,Y 231.783,Z 737.893,A -85,B 0,C 180,E1 10644.735,E2 10644.735} C_VEL
LIN {X 0,Y 226.457,Z 746.741,A -85,B 0,C 180,E1 10641.769,E2 10641.769} C_VEL
LIN {X 0,Y 221.603,Z 753.365,A -85,B 0,C 180,E1 10638.683,E2 10638.683} C_VEL
LIN {X 0,Y 217.291,Z 758.16,A -85,B 0,C 180,E1 10635.478,E2 10635.478} C_VEL
LIN {X 0,Y 213.275,Z 761.414,A -85,B 0,C 180,E1 10631.903,E2 10631.903} C_VEL
LIN {X 0,Y 209.961,Z 762.852,A -85,B 0,C 180,E1 10628.213,E2 10628.213} C_VEL
LIN {X 0,Y 207.193,Z 762.38,A -85,B 0,C 180,E1 10624.15,E2 10624.15} C_VEL
LIN {X 0,Y 205.35,Z 760.064,A -85,B 0,C 180,E1 10620.278,E2 10620.278} C_VEL
LIN {X 0,Y 204.249,Z 756.278,A -85,B 0,C 180,E1 10616.631,E2 10616.631} C_VEL
LIN {X 0,Y 203.669,Z 750.124,A -85,B 0,C 180,E1 10612.602,E2 10612.602} C_VEL
LIN {X 0,Y 203.667,Z 742.605,A -85,B 0,C 180,E1 10608.961,E2 10608.961} C_VEL
LIN {X 0,Y 204.102,Z 733.427,A -85,B 0,C 180,E1 10605.531,E2 10605.531} C_VEL
LIN {X 0,Y 204.484,Z 727.967,A -85,B 0,C 180,E1 10603.816,E2 10603.816} C_VEL
LIN {X 0,Y 205.719,Z 727.769,A -85,B 0,C 180,E1 10602.461,E2 10602.461} C_VEL
LIN {X 0,Y 208.417,Z 726.309,A -85,B 0,C 180,E1 10600.959,E2 10600.959} C_VEL
LIN {X 0,Y 210.741,Z 725.455,A -85,B 0,C 180,E1 10599.445,E2 10599.445} C_VEL
LIN {X 0,Y 213.316,Z 724.115,A -85,B 0,C 180,E1 10598.265,E2 10598.265} C_VEL
LIN {X 0,Y 216.893,Z 722.581,A -85,B 0,C 180,E1 10596.546,E2 10596.546} C_VEL
LIN {X 0,Y 219.584,Z 721.219,A -85,B 0,C 180,E1 10595.52,E2 10595.52} C_VEL
LIN {X 0,Y 224.224,Z 718.974,A -85,B 0,C 180,E1 10593.802,E2 10593.802} C_VEL
LIN {X 0,Y 227.378,Z 717.37,A -85,B 0,C 180,E1 10592.784,E2 10592.784} C_VEL
LIN {X 0,Y 232.77,Z 714.576,A -85,B 0,C 180,E1 10591.242,E2 10591.242} C_VEL
LIN {X 0,Y 242.296,Z 709.281,A -85,B 0,C 180,E1 10588.946,E2 10588.946} C_VEL
LIN {X 0,Y 247.848,Z 705.935,A -85,B 0,C 180,E1 10587.824,E2 10587.824} C_VEL
LIN {X 0,Y 255.464,Z 701.034,A -85,B 0,C 180,E1 10586.504,E2 10586.504} C_VEL
LIN {X 0,Y 259.992,Z 697.833,A -85,B 0,C 180,E1 10585.841,E2 10585.841} C_VEL
LIN {X 0,Y 263.844,Z 695.286,A -85,B 0,C 180,E1 10585.225,E2 10585.225} C_VEL
LIN {X 0,Y 255.653,Z 711.795,A -85,B 0,C 180,E1 10582.722,E2 10582.722} C_VEL
LIN {X 0,Y 247.062,Z 727.245,A -85,B 0,C 180,E1 10579.773,E2 10579.773} C_VEL
LIN {X 0,Y 238.633,Z 741.002,A -85,B 0,C 180,E1 10576.458,E2 10576.458} C_VEL
LIN {X 0,Y 230.351,Z 753.547,A -85,B 0,C 180,E1 10572.621,E2 10572.621} C_VEL
LIN {X 0,Y 222.645,Z 764.621,A -85,B 0,C 180,E1 10568.297,E2 10568.297} C_VEL
LIN {X 0,Y 215.787,Z 774.181,A -85,B 0,C 180,E1 10563.463,E2 10563.463} C_VEL
LIN {X 0,Y 210.053,Z 782.172,A -85,B 0,C 180,E1 10558.115,E2 10558.115} C_VEL
LIN {X 0,Y 205.853,Z 788.256,A -85,B 0,C 180,E1 10552.564,E2 10552.564} C_VEL
LIN {X 0,Y 203.102,Z 792.582,A -85,B 0,C 180,E1 10546.885,E2 10546.885} C_VEL
LIN {X 0,Y 201.613,Z 795.246,A -85,B 0,C 180,E1 10541.152,E2 10541.152} C_VEL
LIN {X 0,Y 201.039,Z 796.312,A -85,B 0,C 180,E1 10535.709,E2 10535.709} C_VEL
LIN {X 0,Y 201.002,Z 795.998,A -85,B 0,C 180,E1 10530.285,E2 10530.285} C_VEL
LIN {X 0,Y 201.489,Z 794.315,A -85,B 0,C 180,E1 10524.875,E2 10524.875} C_VEL
LIN {X 0,Y 202.835,Z 791.004,A -85,B 0,C 180,E1 10519.204,E2 10519.204} C_VEL
LIN {X 0,Y 205.371,Z 786.003,A -85,B 0,C 180,E1 10513.562,E2 10513.562} C_VEL
LIN {X 0,Y 209.228,Z 779.31,A -85,B 0,C 180,E1 10508.115,E2 10508.115} C_VEL
LIN {X 0,Y 214.362,Z 770.964,A -85,B 0,C 180,E1 10502.988,E2 10502.988} C_VEL
LIN {X 0,Y 220.567,Z 761.04,A -85,B 0,C 180,E1 10498.275,E2 10498.275} C_VEL
LIN {X 0,Y 227.712,Z 749.435,A -85,B 0,C 180,E1 10493.958,E2 10493.958} C_VEL
LIN {X 0,Y 235.422,Z 736.333,A -85,B 0,C 180,E1 10490.11,E2 10490.11} C_VEL
LIN {X 0,Y 243.217,Z 722.155,A -85,B 0,C 180,E1 10486.805,E2 10486.805} C_VEL
LIN {X 0,Y 250.815,Z 707.043,A -85,B 0,C 180,E1 10483.982,E2 10483.982} C_VEL
LIN {X 0,Y 258.006,Z 691.14,A -85,B 0,C 180,E1 10481.587,E2 10481.587} C_VEL
LIN {X 0,Y 264.941,Z 673.756,A -85,B 0,C 180,E1 10479.487,E2 10479.487} C_VEL
LIN {X 0,Y 271.09,Z 655.743,A -85,B 0,C 180,E1 10477.754,E2 10477.754} C_VEL
LIN {X 0,Y 276.584,Z 636.214,A -85,B 0,C 180,E1 10476.278,E2 10476.278} C_VEL
LIN {X 0,Y 281.134,Z 615.31,A -85,B 0,C 180,E1 10475.081,E2 10475.081} C_VEL
LIN {X 0,Y 287.684,Z 581.452,A -85,B 0,C 180,E1 10473.585,E2 10473.585} C_VEL
LIN {X 0,Y 282.035,Z 592.662,A -85,B 0,C 180,E1 10472.758,E2 10472.758} C_VEL
LIN {X 0,Y 280.499,Z 596.044,A -85,B 0,C 180,E1 10472.566,E2 10472.566} C_VEL
LIN {X 0,Y 278.995,Z 599.669,A -85,B 0,C 180,E1 10472.426,E2 10472.426} C_VEL
LIN {X 0,Y 277.052,Z 605.471,A -85,B 0,C 180,E1 10472.397,E2 10472.397} C_VEL
LIN {X 0,Y 273.975,Z 617.24,A -85,B 0,C 180,E1 10472.696,E2 10472.696} C_VEL
LIN {X 0,Y 271.936,Z 621.903,A -85,B 0,C 180,E1 10472.535,E2 10472.535} C_VEL
LIN {X 0,Y 271.58,Z 622.493,A -85,B 0,C 180,E1 10472.48,E2 10472.48} C_VEL
LIN {X 0,Y 269.892,Z 625.443,A -85,B 0,C 180,E1 10472.241,E2 10472.241} C_VEL
LIN {X 0,Y 264.234,Z 636.061,A -85,B 0,C 180,E1 10471.595,E2 10471.595} C_VEL
LIN {X 0,Y 258.476,Z 644.775,A -85,B 0,C 180,E1 10470.706,E2 10470.706} C_VEL
LIN {X 0,Y 256.397,Z 647.683,A -85,B 0,C 180,E1 10470.376,E2 10470.376} C_VEL
LIN {X 0,Y 250.683,Z 656.398,A -85,B 0,C 180,E1 10469.643,E2 10469.643} C_VEL
LIN {X 0,Y 244.696,Z 663.978,A -85,B 0,C 180,E1 10468.561,E2 10468.561} C_VEL
LIN {X 0,Y 241.036,Z 668.077,A -85,B 0,C 180,E1 10467.806,E2 10467.806} C_VEL
LIN {X 0,Y 234.994,Z 675.423,A -85,B 0,C 180,E1 10466.681,E2 10466.681} C_VEL
LIN {X 0,Y 230.137,Z 680.287,A -85,B 0,C 180,E1 10465.476,E2 10465.476} C_VEL
LIN {X 0,Y 227.723,Z 682.665,A -85,B 0,C 180,E1 10464.792,E2 10464.792} C_VEL
LIN {X 0,Y 222.277,Z 688.448,A -85,B 0,C 180,E1 10463.415,E2 10463.415} C_VEL
LIN {X 0,Y 217.357,Z 692.873,A -85,B 0,C 180,E1 10461.686,E2 10461.686} C_VEL
LIN {X 0,Y 213.127,Z 697.167,A -85,B 0,C 180,E1 10460.315,E2 10460.315} C_VEL
LIN {X 0,Y 208.98,Z 700.709,A -85,B 0,C 180,E1 10458.409,E2 10458.409} C_VEL
LIN {X 0,Y 205.408,Z 704.229,A -85,B 0,C 180,E1 10456.982,E2 10456.982} C_VEL
LIN {X 0,Y 202.948,Z 706.334,A -85,B 0,C 180,E1 10455.43,E2 10455.43} C_VEL
LIN {X 0,Y 202.011,Z 707.252,A -85,B 0,C 180,E1 10454.915,E2 10454.915} C_VEL
LIN {X 0,Y 199.069,Z 710.324,A -85,B 0,C 180,E1 10453.36,E2 10453.36} C_VEL
LIN {X 0,Y 197.644,Z 711.565,A -85,B 0,C 180,E1 10451.972,E2 10451.972} C_VEL
LIN {X 0,Y 197.514,Z 711.868,A -85,B 0,C 180,E1 10451.684,E2 10451.684} C_VEL
LIN {X 0,Y 196.43,Z 724.657,A -85,B 0,C 180,E1 10448.195,E2 10448.195} C_VEL
LIN {X 0,Y 195.749,Z 735.942,A -85,B 0,C 180,E1 10444.395,E2 10444.395} C_VEL
LIN {X 0,Y 195.554,Z 745.72,A -85,B 0,C 180,E1 10440.294,E2 10440.294} C_VEL
LIN {X 0,Y 195.996,Z 753.905,A -85,B 0,C 180,E1 10435.906,E2 10435.906} C_VEL
LIN {X 0,Y 197.16,Z 760.028,A -85,B 0,C 180,E1 10431.544,E2 10431.544} C_VEL
LIN {X 0,Y 199.141,Z 764.361,A -85,B 0,C 180,E1 10427.238,E2 10427.238} C_VEL
LIN {X 0,Y 202.23,Z 767,A -85,B 0,C 180,E1 10422.745,E2 10422.745} C_VEL
LIN {X 0,Y 206.071,Z 767.78,A -85,B 0,C 180,E1 10418.661,E2 10418.661} C_VEL
LIN {X 0,Y 211.533,Z 766.613,A -85,B 0,C 180,E1 10414.225,E2 10414.225} C_VEL
LIN {X 0,Y 217.307,Z 763.826,A -85,B 0,C 180,E1 10410.508,E2 10410.508} C_VEL
LIN {X 0,Y 224.42,Z 758.999,A -85,B 0,C 180,E1 10406.771,E2 10406.771} C_VEL
LIN {X 0,Y 232.46,Z 752.157,A -85,B 0,C 180,E1 10403.284,E2 10403.284} C_VEL
LIN {X 0,Y 235.683,Z 749.303,A -85,B 0,C 180,E1 10402.051,E2 10402.051} C_VEL
LIN {X 0,Y 227.466,Z 763.995,A -85,B 0,C 180,E1 10398.734,E2 10398.734} C_VEL
LIN {X 0,Y 219.51,Z 777.409,A -85,B 0,C 180,E1 10394.912,E2 10394.912} C_VEL
LIN {X 0,Y 211.701,Z 790.179,A -85,B 0,C 180,E1 10390.32,E2 10390.32} C_VEL
LIN {X 0,Y 205.206,Z 800.833,A -85,B 0,C 180,E1 10385.438,E2 10385.438} C_VEL
LIN {X 0,Y 199.599,Z 810.462,A -85,B 0,C 180,E1 10379.731,E2 10379.731} C_VEL
LIN {X 0,Y 195.715,Z 818.161,A -85,B 0,C 180,E1 10373.803,E2 10373.803} C_VEL
LIN {X 0,Y 193.457,Z 824.045,A -85,B 0,C 180,E1 10367.754,E2 10367.754} C_VEL
LIN {X 0,Y 192.591,Z 828.207,A -85,B 0,C 180,E1 10361.682,E2 10361.682} C_VEL
LIN {X 0,Y 192.643,Z 830.673,A -85,B 0,C 180,E1 10355.958,E2 10355.958} C_VEL
LIN {X 0,Y 192.82,Z 831.638,A -85,B 0,C 180,E1 10351.188,E2 10351.188} C_VEL
LIN {X 0,Y 192.724,Z 831.558,A -85,B 0,C 180,E1 10346.431,E2 10346.431} C_VEL
LIN {X 0,Y 192.503,Z 830.329,A -85,B 0,C 180,E1 10341.337,E2 10341.337} C_VEL
LIN {X 0,Y 192.824,Z 827.477,A -85,B 0,C 180,E1 10335.281,E2 10335.281} C_VEL
LIN {X 0,Y 194.494,Z 822.744,A -85,B 0,C 180,E1 10328.908,E2 10328.908} C_VEL
LIN {X 0,Y 198.105,Z 815.85,A -85,B 0,C 180,E1 10322.333,E2 10322.333} C_VEL
LIN {X 0,Y 203.197,Z 807.729,A -85,B 0,C 180,E1 10316.556,E2 10316.556} C_VEL
LIN {X 0,Y 210.019,Z 797.579,A -85,B 0,C 180,E1 10311.065,E2 10311.065} C_VEL
LIN {X 0,Y 218.034,Z 785.869,A -85,B 0,C 180,E1 10306.175,E2 10306.175} C_VEL
LIN {X 0,Y 226.406,Z 773.375,A -85,B 0,C 180,E1 10302.104,E2 10302.104} C_VEL
LIN {X 0,Y 235.776,Z 758.536,A -85,B 0,C 180,E1 10298.322,E2 10298.322} C_VEL
LIN {X 0,Y 245.322,Z 742.195,A -85,B 0,C 180,E1 10295.076,E2 10295.076} C_VEL
LIN {X 0,Y 254.128,Z 725.466,A -85,B 0,C 180,E1 10292.478,E2 10292.478} C_VEL
LIN {X 0,Y 256.057,Z 721.492,A -85,B 0,C 180,E1 10291.945,E2 10291.945} C_VEL
LIN {X 0,Y 243.994,Z 728.667,A -85,B 0,C 180,E1 10290.267,E2 10290.267} C_VEL
LIN {X 0,Y 236.029,Z 732.623,A -85,B 0,C 180,E1 10288.876,E2 10288.876} C_VEL
LIN {X 0,Y 229.524,Z 735.532,A -85,B 0,C 180,E1 10287.5,E2 10287.5} C_VEL
LIN {X 0,Y 223.545,Z 745.252,A -85,B 0,C 180,E1 10284.579,E2 10284.579} C_VEL
LIN {X 0,Y 218.034,Z 752.626,A -85,B 0,C 180,E1 10281.521,E2 10281.521} C_VEL
LIN {X 0,Y 213.076,Z 758.108,A -85,B 0,C 180,E1 10278.323,E2 10278.323} C_VEL
LIN {X 0,Y 208.37,Z 762.076,A -85,B 0,C 180,E1 10274.732,E2 10274.732} C_VEL
LIN {X 0,Y 204.378,Z 764.174,A -85,B 0,C 180,E1 10270.998,E2 10270.998} C_VEL
LIN {X 0,Y 201.139,Z 764.494,A -85,B 0,C 180,E1 10267.138,E2 10267.138} C_VEL
LIN {X 0,Y 198.67,Z 763.052,A -85,B 0,C 180,E1 10263.172,E2 10263.172} C_VEL
LIN {X 0,Y 196.959,Z 759.799,A -85,B 0,C 180,E1 10259.126,E2 10259.126} C_VEL
LIN {X 0,Y 195.96,Z 754.63,A -85,B 0,C 180,E1 10255.023,E2 10255.023} C_VEL
LIN {X 0,Y 195.622,Z 747.908,A -85,B 0,C 180,E1 10251.179,E2 10251.179} C_VEL
LIN {X 0,Y 195.787,Z 739.804,A -85,B 0,C 180,E1 10247.613,E2 10247.613} C_VEL
LIN {X 0,Y 196.053,Z 735.273,A -85,B 0,C 180,E1 10245.829,E2 10245.829} C_VEL
LIN {X 0,Y 197.136,Z 735.037,A -85,B 0,C 180,E1 10244.405,E2 10244.405} C_VEL
LIN {X 0,Y 199.491,Z 733.789,A -85,B 0,C 180,E1 10242.799,E2 10242.799} C_VEL
LIN {X 0,Y 201.974,Z 732.854,A -85,B 0,C 180,E1 10240.929,E2 10240.929} C_VEL
LIN {X 0,Y 203.841,Z 731.942,A -85,B 0,C 180,E1 10239.917,E2 10239.917} C_VEL
LIN {X 0,Y 206.911,Z 730.726,A -85,B 0,C 180,E1 10238.154,E2 10238.154} C_VEL
LIN {X 0,Y 209.472,Z 729.578,A -85,B 0,C 180,E1 10236.957,E2 10236.957} C_VEL
LIN {X 0,Y 213.921,Z 727.605,A -85,B 0,C 180,E1 10235.061,E2 10235.061} C_VEL
LIN {X 0,Y 221.011,Z 724.348,A -85,B 0,C 180,E1 10232.518,E2 10232.518} C_VEL
LIN {X 0,Y 229.712,Z 720.158,A -85,B 0,C 180,E1 10230.019,E2 10230.019} C_VEL
LIN {X 0,Y 240.54,Z 714.393,A -85,B 0,C 180,E1 10227.546,E2 10227.546} C_VEL
LIN {X 0,Y 252.194,Z 707.624,A -85,B 0,C 180,E1 10225.462,E2 10225.462} C_VEL
LIN {X 0,Y 254.034,Z 706.54,A -85,B 0,C 180,E1 10225.15,E2 10225.15} C_VEL
LIN {X 0,Y 245.075,Z 722.618,A -85,B 0,C 180,E1 10222.325,E2 10222.325} C_VEL
LIN {X 0,Y 235.853,Z 737.488,A -85,B 0,C 180,E1 10218.991,E2 10218.991} C_VEL
LIN {X 0,Y 226.739,Z 750.95,A -85,B 0,C 180,E1 10215.124,E2 10215.124} C_VEL
LIN {X 0,Y 218.454,Z 762.414,A -85,B 0,C 180,E1 10210.883,E2 10210.883} C_VEL
LIN {X 0,Y 210.819,Z 772.54,A -85,B 0,C 180,E1 10206.023,E2 10206.023} C_VEL
LIN {X 0,Y 204.295,Z 781.077,A -85,B 0,C 180,E1 10200.597,E2 10200.597} C_VEL
LIN {X 0,Y 199.214,Z 787.82,A -85,B 0,C 180,E1 10194.706,E2 10194.706} C_VEL
LIN {X 0,Y 195.854,Z 792.565,A -85,B 0,C 180,E1 10188.761,E2 10188.761} C_VEL
LIN {X 0,Y 193.966,Z 795.564,A -85,B 0,C 180,E1 10182.807,E2 10182.807} C_VEL
LIN {X 0,Y 193.166,Z 796.959,A -85,B 0,C 180,E1 10177.136,E2 10177.136} C_VEL
LIN {X 0,Y 193.004,Z 796.929,A -85,B 0,C 180,E1 10171.484,E2 10171.484} C_VEL
LIN {X 0,Y 193.349,Z 795.619,A -85,B 0,C 180,E1 10166.145,E2 10166.145} C_VEL
LIN {X 0,Y 194.53,Z 792.724,A -85,B 0,C 180,E1 10160.235,E2 10160.235} C_VEL
LIN {X 0,Y 196.881,Z 788.21,A -85,B 0,C 180,E1 10154.386,E2 10154.386} C_VEL
LIN {X 0,Y 200.653,Z 781.979,A -85,B 0,C 180,E1 10148.669,E2 10148.669} C_VEL
LIN {X 0,Y 205.618,Z 774.332,A -85,B 0,C 180,E1 10143.425,E2 10143.425} C_VEL
LIN {X 0,Y 211.937,Z 764.829,A -85,B 0,C 180,E1 10138.421,E2 10138.421} C_VEL
LIN {X 0,Y 219.125,Z 753.869,A -85,B 0,C 180,E1 10133.941,E2 10133.941} C_VEL
LIN {X 0,Y 226.918,Z 741.492,A -85,B 0,C 180,E1 10129.96,E2 10129.96} C_VEL
LIN {X 0,Y 235.335,Z 727.179,A -85,B 0,C 180,E1 10126.337,E2 10126.337} C_VEL
LIN {X 0,Y 243.557,Z 711.865,A -85,B 0,C 180,E1 10123.282,E2 10123.282} C_VEL
LIN {X 0,Y 251.205,Z 696.011,A -85,B 0,C 180,E1 10120.751,E2 10120.751} C_VEL
LIN {X 0,Y 258.415,Z 679.136,A -85,B 0,C 180,E1 10118.594,E2 10118.594} C_VEL
LIN {X 0,Y 265.232,Z 660.517,A -85,B 0,C 180,E1 10116.705,E2 10116.705} C_VEL
LIN {X 0,Y 271.012,Z 641.489,A -85,B 0,C 180,E1 10115.195,E2 10115.195} C_VEL
LIN {X 0,Y 275.638,Z 622.339,A -85,B 0,C 180,E1 10114.017,E2 10114.017} C_VEL
LIN {X 0,Y 277.908,Z 610.979,A -85,B 0,C 180,E1 10113.416,E2 10113.416} C_VEL
LIN {X 0,Y 272.119,Z 621.631,A -85,B 0,C 180,E1 10112.568,E2 10112.568} C_VEL
LIN {X 0,Y 271.58,Z 622.493,A -85,B 0,C 180,E1 10112.48,E2 10112.48} C_VEL
LIN {X 0,Y 268.583,Z 628.039,A -85,B 0,C 180,E1 10112.092,E2 10112.092} C_VEL
LIN {X 0,Y 265.068,Z 636.115,A -85,B 0,C 180,E1 10111.957,E2 10111.957} C_VEL
LIN {X 0,Y 259.136,Z 649.338,A -85,B 0,C 180,E1 10111.948,E2 10111.948} C_VEL
LIN {X 0,Y 256.325,Z 654.022,A -85,B 0,C 180,E1 10111.751,E2 10111.751} C_VEL
LIN {X 0,Y 249.476,Z 663.362,A -85,B 0,C 180,E1 10110.865,E2 10110.865} C_VEL
LIN {X 0,Y 243.449,Z 670.164,A -85,B 0,C 180,E1 10109.8,E2 10109.8} C_VEL
LIN {X 0,Y 240.818,Z 673.159,A -85,B 0,C 180,E1 10109.318,E2 10109.318} C_VEL
LIN {X 0,Y 234.527,Z 680.189,A -85,B 0,C 180,E1 10108.245,E2 10108.245} C_VEL
LIN {X 0,Y 228.66,Z 685.825,A -85,B 0,C 180,E1 10106.87,E2 10106.87} C_VEL
LIN {X 0,Y 226.085,Z 688.239,A -85,B 0,C 180,E1 10106.249,E2 10106.249} C_VEL
LIN {X 0,Y 220.387,Z 693.887,A -85,B 0,C 180,E1 10104.855,E2 10104.855} C_VEL
LIN {X 0,Y 215.429,Z 698.03,A -85,B 0,C 180,E1 10103.236,E2 10103.236} C_VEL
LIN {X 0,Y 210.516,Z 702.573,A -85,B 0,C 180,E1 10101.745,E2 10101.745} C_VEL
LIN {X 0,Y 206.129,Z 706.195,A -85,B 0,C 180,E1 10099.85,E2 10099.85} C_VEL
LIN {X 0,Y 201.846,Z 709.996,A -85,B 0,C 180,E1 10098.185,E2 10098.185} C_VEL
LIN {X 0,Y 198.699,Z 712.519,A -85,B 0,C 180,E1 10096.368,E2 10096.368} C_VEL
LIN {X 0,Y 195.085,Z 715.935,A -85,B 0,C 180,E1 10094.546,E2 10094.546} C_VEL
LIN {X 0,Y 193.123,Z 717.581,A -85,B 0,C 180,E1 10092.864,E2 10092.864} C_VEL
LIN {X 0,Y 190.312,Z 720.434,A -85,B 0,C 180,E1 10091.21,E2 10091.21} C_VEL
LIN {X 0,Y 188.758,Z 721.922,A -85,B 0,C 180,E1 10089.452,E2 10089.452} C_VEL
LIN {X 0,Y 188.633,Z 722.261,A -85,B 0,C 180,E1 10089.074,E2 10089.074} C_VEL
LIN {X 0,Y 187.845,Z 734.051,A -85,B 0,C 180,E1 10085.193,E2 10085.193} C_VEL
LIN {X 0,Y 187.551,Z 743.886,A -85,B 0,C 180,E1 10081.223,E2 10081.223} C_VEL
LIN {X 0,Y 187.874,Z 752.882,A -85,B 0,C 180,E1 10076.645,E2 10076.645} C_VEL
LIN {X 0,Y 188.958,Z 759.724,A -85,B 0,C 180,E1 10072.093,E2 10072.093} C_VEL
LIN {X 0,Y 190.895,Z 764.743,A -85,B 0,C 180,E1 10067.6,E2 10067.6} C_VEL
LIN {X 0,Y 194.245,Z 768.294,A -85,B 0,C 180,E1 10062.631,E2 10062.631} C_VEL
LIN {X 0,Y 198.522,Z 769.641,A -85,B 0,C 180,E1 10058.119,E2 10058.119} C_VEL
LIN {X 0,Y 204.036,Z 769.162,A -85,B 0,C 180,E1 10053.738,E2 10053.738} C_VEL
LIN {X 0,Y 210.83,Z 766.667,A -85,B 0,C 180,E1 10049.507,E2 10049.507} C_VEL
LIN {X 0,Y 218.374,Z 762.379,A -85,B 0,C 180,E1 10045.726,E2 10045.726} C_VEL
LIN {X 0,Y 226.88,Z 756.248,A -85,B 0,C 180,E1 10042.225,E2 10042.225} C_VEL
LIN {X 0,Y 224.829,Z 758.11,A -85,B 0,C 180,E1 10041.51,E2 10041.51} C_VEL
LIN {X 0,Y 215.65,Z 773.174,A -85,B 0,C 180,E1 10037.494,E2 10037.494} C_VEL
LIN {X 0,Y 207.535,Z 785.823,A -85,B 0,C 180,E1 10033.167,E2 10033.167} C_VEL
LIN {X 0,Y 200.218,Z 797.042,A -85,B 0,C 180,E1 10028.261,E2 10028.261} C_VEL
LIN {X 0,Y 194.02,Z 806.867,A -85,B 0,C 180,E1 10022.759,E2 10022.759} C_VEL
LIN {X 0,Y 189.24,Z 815.19,A -85,B 0,C 180,E1 10016.686,E2 10016.686} C_VEL
LIN {X 0,Y 186.119,Z 821.886,A -85,B 0,C 180,E1 10010.11,E2 10010.11} C_VEL
LIN {X 0,Y 184.761,Z 826.536,A -85,B 0,C 180,E1 10003.775,E2 10003.775} C_VEL
LIN {X 0,Y 184.592,Z 829.432,A -85,B 0,C 180,E1 9997.783,E2 9997.783} C_VEL
LIN {X 0,Y 184.808,Z 830.711,A -85,B 0,C 180,E1 9992.791,E2 9992.791} C_VEL
LIN {X 0,Y 184.824,Z 830.983,A -85,B 0,C 180,E1 9988.14,E2 9988.14} C_VEL
LIN {X 0,Y 184.593,Z 830.277,A -85,B 0,C 180,E1 9983.156,E2 9983.156} C_VEL
LIN {X 0,Y 184.633,Z 828.06,A -85,B 0,C 180,E1 9977.098,E2 9977.098} C_VEL
LIN {X 0,Y 185.89,Z 824.021,A -85,B 0,C 180,E1 9970.519,E2 9970.519} C_VEL
LIN {X 0,Y 189.085,Z 817.866,A -85,B 0,C 180,E1 9963.629,E2 9963.629} C_VEL
LIN {X 0,Y 194.139,Z 810.031,A -85,B 0,C 180,E1 9957.263,E2 9957.263} C_VEL
LIN {X 0,Y 201.071,Z 800.244,A -85,B 0,C 180,E1 9951.324,E2 9951.324} C_VEL
LIN {X 0,Y 209.235,Z 789.047,A -85,B 0,C 180,E1 9946.139,E2 9946.139} C_VEL
LIN {X 0,Y 218.328,Z 776.247,A -85,B 0,C 180,E1 9941.608,E2 9941.608} C_VEL
LIN {X 0,Y 227.716,Z 762.339,A -85,B 0,C 180,E1 9937.781,E2 9937.781} C_VEL
LIN {X 0,Y 237.346,Z 746.968,A -85,B 0,C 180,E1 9934.477,E2 9934.477} C_VEL
LIN {X 0,Y 245.507,Z 732.63,A -85,B 0,C 180,E1 9932.029,E2 9932.029} C_VEL
LIN {X 0,Y 234.243,Z 738.059,A -85,B 0,C 180,E1 9930.243,E2 9930.243} C_VEL
LIN {X 0,Y 224.08,Z 742.231,A -85,B 0,C 180,E1 9928.227,E2 9928.227} C_VEL
LIN {X 0,Y 221.852,Z 742.961,A -85,B 0,C 180,E1 9927.658,E2 9927.658} C_VEL
LIN {X 0,Y 215.897,Z 750.898,A -85,B 0,C 180,E1 9924.808,E2 9924.808} C_VEL
LIN {X 0,Y 209.936,Z 757.532,A -85,B 0,C 180,E1 9921.513,E2 9921.513} C_VEL
LIN {X 0,Y 204.08,Z 762.558,A -85,B 0,C 180,E1 9917.682,E2 9917.682} C_VEL
LIN {X 0,Y 199.054,Z 765.429,A -85,B 0,C 180,E1 9913.654,E2 9913.654} C_VEL
LIN {X 0,Y 194.93,Z 766.277,A -85,B 0,C 180,E1 9909.446,E2 9909.446} C_VEL
LIN {X 0,Y 191.924,Z 765.25,A -85,B 0,C 180,E1 9905.38,E2 9905.38} C_VEL
LIN {X 0,Y 189.741,Z 762.462,A -85,B 0,C 180,E1 9901.207,E2 9901.207} C_VEL
LIN {X 0,Y 188.354,Z 757.823,A -85,B 0,C 180,E1 9896.956,E2 9896.956} C_VEL
LIN {X 0,Y 187.698,Z 751.116,A -85,B 0,C 180,E1 9892.654,E2 9892.654} C_VEL
LIN {X 0,Y 187.725,Z 742.19,A -85,B 0,C 180,E1 9888.322,E2 9888.322} C_VEL
LIN {X 0,Y 188.819,Z 741.855,A -85,B 0,C 180,E1 9886.525,E2 9886.525} C_VEL
LIN {X 0,Y 190.583,Z 740.861,A -85,B 0,C 180,E1 9885.103,E2 9885.103} C_VEL
LIN {X 0,Y 192.59,Z 740.148,A -85,B 0,C 180,E1 9883.097,E2 9883.097} C_VEL
LIN {X 0,Y 194.574,Z 739.234,A -85,B 0,C 180,E1 9881.731,E2 9881.731} C_VEL
LIN {X 0,Y 197.844,Z 737.931,A -85,B 0,C 180,E1 9879.59,E2 9879.59} C_VEL
LIN {X 0,Y 203.065,Z 735.838,A -85,B 0,C 180,E1 9876.801,E2 9876.801} C_VEL
LIN {X 0,Y 209.62,Z 733.12,A -85,B 0,C 180,E1 9873.97,E2 9873.97} C_VEL
LIN {X 0,Y 217.787,Z 729.58,A -85,B 0,C 180,E1 9871.179,E2 9871.179} C_VEL
LIN {X 0,Y 226.914,Z 725.395,A -85,B 0,C 180,E1 9868.67,E2 9868.67} C_VEL
LIN {X 0,Y 238.175,Z 719.755,A -85,B 0,C 180,E1 9866.224,E2 9866.224} C_VEL
LIN {X 0,Y 244.29,Z 716.482,A -85,B 0,C 180,E1 9865.123,E2 9865.123} C_VEL
LIN {X 0,Y 235.335,Z 731.037,A -85,B 0,C 180,E1 9862.21,E2 9862.21} C_VEL
LIN {X 0,Y 226.091,Z 744.676,A -85,B 0,C 180,E1 9858.747,E2 9858.747} C_VEL
LIN {X 0,Y 217.163,Z 756.865,A -85,B 0,C 180,E1 9854.785,E2 9854.785} C_VEL
LIN {X 0,Y 208.37,Z 768.144,A -85,B 0,C 180,E1 9850.016,E2 9850.016} C_VEL
LIN {X 0,Y 200.952,Z 777.303,A -85,B 0,C 180,E1 9844.904,E2 9844.904} C_VEL
LIN {X 0,Y 194.727,Z 784.923,A -85,B 0,C 180,E1 9839.196,E2 9839.196} C_VEL
LIN {X 0,Y 190.166,Z 790.669,A -85,B 0,C 180,E1 9833.225,E2 9833.225} C_VEL
LIN {X 0,Y 187.094,Z 794.833,A -85,B 0,C 180,E1 9826.773,E2 9826.773} C_VEL
LIN {X 0,Y 185.588,Z 797.116,A -85,B 0,C 180,E1 9820.555,E2 9820.555} C_VEL
LIN {X 0,Y 185.06,Z 797.825,A -85,B 0,C 180,E1 9814.649,E2 9814.649} C_VEL
LIN {X 0,Y 185.134,Z 797.215,A -85,B 0,C 180,E1 9809.072,E2 9809.072} C_VEL
LIN {X 0,Y 185.834,Z 795.262,A -85,B 0,C 180,E1 9803.202,E2 9803.202} C_VEL
LIN {X 0,Y 187.63,Z 791.682,A -85,B 0,C 180,E1 9797.067,E2 9797.067} C_VEL
LIN {X 0,Y 191.02,Z 786.14,A -85,B 0,C 180,E1 9790.746,E2 9790.746} C_VEL
LIN {X 0,Y 195.821,Z 779.039,A -85,B 0,C 180,E1 9784.925,E2 9784.925} C_VEL
LIN {X 0,Y 201.836,Z 770.474,A -85,B 0,C 180,E1 9779.649,E2 9779.649} C_VEL
LIN {X 0,Y 208.805,Z 760.54,A -85,B 0,C 180,E1 9774.927,E2 9774.927} C_VEL
LIN {X 0,Y 216.929,Z 748.591,A -85,B 0,C 180,E1 9770.501,E2 9770.501} C_VEL
LIN {X 0,Y 225.57,Z 735.048,A -85,B 0,C 180,E1 9766.602,E2 9766.602} C_VEL
LIN {X 0,Y 234.185,Z 720.351,A -85,B 0,C 180,E1 9763.284,E2 9763.284} C_VEL
LIN {X 0,Y 242.521,Z 704.644,A -85,B 0,C 180,E1 9760.478,E2 9760.478} C_VEL
LIN {X 0,Y 250.348,Z 688.005,A -85,B 0,C 180,E1 9758.113,E2 9758.113} C_VEL
LIN {X 0,Y 257.5,Z 670.507,A -85,B 0,C 180,E1 9756.132,E2 9756.132} C_VEL
LIN {X 0,Y 263.852,Z 652.183,A -85,B 0,C 180,E1 9754.491,E2 9754.491} C_VEL
LIN {X 0,Y 268.463,Z 635.986,A -85,B 0,C 180,E1 9753.323,E2 9753.323} C_VEL
LIN {X 0,Y 262.079,Z 645.918,A -85,B 0,C 180,E1 9752.526,E2 9752.526} C_VEL
LIN {X 0,Y 257.939,Z 651.611,A -85,B 0,C 180,E1 9751.905,E2 9751.905} C_VEL
LIN {X 0,Y 256.325,Z 654.022,A -85,B 0,C 180,E1 9751.751,E2 9751.751} C_VEL
LIN {X 0,Y 253.232,Z 659.283,A -85,B 0,C 180,E1 9751.589,E2 9751.589} C_VEL
LIN {X 0,Y 247.809,Z 669.4,A -85,B 0,C 180,E1 9751.724,E2 9751.724} C_VEL
LIN {X 0,Y 244.835,Z 673.525,A -85,B 0,C 180,E1 9751.528,E2 9751.528} C_VEL
LIN {X 0,Y 243.923,Z 674.509,A -85,B 0,C 180,E1 9751.39,E2 9751.39} C_VEL
LIN {X 0,Y 240.698,Z 677.955,A -85,B 0,C 180,E1 9750.866,E2 9750.866} C_VEL
LIN {X 0,Y 233.753,Z 685.285,A -85,B 0,C 180,E1 9749.749,E2 9749.749} C_VEL
LIN {X 0,Y 227.022,Z 691.402,A -85,B 0,C 180,E1 9748.254,E2 9748.254} C_VEL
LIN {X 0,Y 218.487,Z 699.126,A -85,B 0,C 180,E1 9746.354,E2 9746.354} C_VEL
LIN {X 0,Y 213.014,Z 703.586,A -85,B 0,C 180,E1 9744.694,E2 9744.694} C_VEL
LIN {X 0,Y 207.283,Z 708.384,A -85,B 0,C 180,E1 9743,E2 9743} C_VEL
LIN {X 0,Y 202.544,Z 712.08,A -85,B 0,C 180,E1 9741.124,E2 9741.124} C_VEL
LIN {X 0,Y 197.701,Z 716.042,A -85,B 0,C 180,E1 9739.193,E2 9739.193} C_VEL
LIN {X 0,Y 194.772,Z 718.223,A -85,B 0,C 180,E1 9737.632,E2 9737.632} C_VEL
LIN {X 0,Y 190.608,Z 721.752,A -85,B 0,C 180,E1 9735.518,E2 9735.518} C_VEL
LIN {X 0,Y 188.555,Z 723.383,A -85,B 0,C 180,E1 9733.973,E2 9733.973} C_VEL
LIN {X 0,Y 185.58,Z 726.183,A -85,B 0,C 180,E1 9732.131,E2 9732.131} C_VEL
LIN {X 0,Y 183.536,Z 728.017,A -85,B 0,C 180,E1 9730.041,E2 9730.041} C_VEL
LIN {X 0,Y 180.936,Z 730.682,A -85,B 0,C 180,E1 9727.942,E2 9727.942} C_VEL
LIN {X 0,Y 179.958,Z 732.057,A -85,B 0,C 180,E1 9725.989,E2 9725.989} C_VEL
LIN {X 0,Y 179.564,Z 742.343,A -85,B 0,C 180,E1 9721.916,E2 9721.916} C_VEL
LIN {X 0,Y 179.761,Z 751.488,A -85,B 0,C 180,E1 9717.451,E2 9717.451} C_VEL
LIN {X 0,Y 180.745,Z 759.093,A -85,B 0,C 180,E1 9712.691,E2 9712.691} C_VEL
LIN {X 0,Y 182.626,Z 764.821,A -85,B 0,C 180,E1 9707.993,E2 9707.993} C_VEL
LIN {X 0,Y 185.984,Z 769.174,A -85,B 0,C 180,E1 9702.803,E2 9702.803} C_VEL
LIN {X 0,Y 190.345,Z 771.275,A -85,B 0,C 180,E1 9698.103,E2 9698.103} C_VEL
LIN {X 0,Y 195.894,Z 771.6,A -85,B 0,C 180,E1 9693.638,E2 9693.638} C_VEL
LIN {X 0,Y 203.02,Z 769.95,A -85,B 0,C 180,E1 9689.191,E2 9689.191} C_VEL
LIN {X 0,Y 210.83,Z 766.59,A -85,B 0,C 180,E1 9685.314,E2 9685.314} C_VEL
LIN {X 0,Y 217.876,Z 762.567,A -85,B 0,C 180,E1 9682.338,E2 9682.338} C_VEL
LIN {X 0,Y 214.463,Z 765.25,A -85,B 0,C 180,E1 9681.131,E2 9681.131} C_VEL
LIN {X 0,Y 205.386,Z 779.06,A -85,B 0,C 180,E1 9676.906,E2 9676.906} C_VEL
LIN {X 0,Y 196.991,Z 791.296,A -85,B 0,C 180,E1 9672.066,E2 9672.066} C_VEL
LIN {X 0,Y 189.643,Z 802.038,A -85,B 0,C 180,E1 9666.568,E2 9666.568} C_VEL
LIN {X 0,Y 183.945,Z 810.802,A -85,B 0,C 180,E1 9660.727,E2 9660.727} C_VEL
LIN {X 0,Y 179.704,Z 818.23,A -85,B 0,C 180,E1 9654.152,E2 9654.152} C_VEL
LIN {X 0,Y 177.343,Z 823.856,A -85,B 0,C 180,E1 9647.386,E2 9647.386} C_VEL
LIN {X 0,Y 176.592,Z 827.646,A -85,B 0,C 180,E1 9640.769,E2 9640.769} C_VEL
LIN {X 0,Y 176.745,Z 829.64,A -85,B 0,C 180,E1 9634.868,E2 9634.868} C_VEL
LIN {X 0,Y 176.905,Z 830.262,A -85,B 0,C 180,E1 9630,E2 9630} C_VEL
LIN {X 0,Y 176.7,Z 829.93,A -85,B 0,C 180,E1 9624.798,E2 9624.798} C_VEL
LIN {X 0,Y 176.554,Z 828.328,A -85,B 0,C 180,E1 9618.898,E2 9618.898} C_VEL
LIN {X 0,Y 177.464,Z 824.838,A -85,B 0,C 180,E1 9611.948,E2 9611.948} C_VEL
LIN {X 0,Y 180.129,Z 819.614,A -85,B 0,C 180,E1 9605.047,E2 9605.047} C_VEL
LIN {X 0,Y 184.826,Z 812.51,A -85,B 0,C 180,E1 9598.349,E2 9598.349} C_VEL
LIN {X 0,Y 191.646,Z 803.336,A -85,B 0,C 180,E1 9591.979,E2 9591.979} C_VEL
LIN {X 0,Y 199.605,Z 793.052,A -85,B 0,C 180,E1 9586.578,E2 9586.578} C_VEL
LIN {X 0,Y 208.901,Z 780.82,A -85,B 0,C 180,E1 9581.697,E2 9581.697} C_VEL
LIN {X 0,Y 219.065,Z 766.78,A -85,B 0,C 180,E1 9577.422,E2 9577.422} C_VEL
LIN {X 0,Y 229.026,Z 752.012,A -85,B 0,C 180,E1 9573.953,E2 9573.953} C_VEL
LIN {X 0,Y 234.923,Z 742.348,A -85,B 0,C 180,E1 9572.069,E2 9572.069} C_VEL
LIN {X 0,Y 221.949,Z 747.409,A -85,B 0,C 180,E1 9569.704,E2 9569.704} C_VEL
LIN {X 0,Y 213.796,Z 749.984,A -85,B 0,C 180,E1 9567.731,E2 9567.731} C_VEL
LIN {X 0,Y 207.14,Z 757.201,A -85,B 0,C 180,E1 9564.526,E2 9564.526} C_VEL
LIN {X 0,Y 200.458,Z 762.9,A -85,B 0,C 180,E1 9560.74,E2 9560.74} C_VEL
LIN {X 0,Y 194.605,Z 766.427,A -85,B 0,C 180,E1 9556.72,E2 9556.72} C_VEL
LIN {X 0,Y 189.671,Z 767.924,A -85,B 0,C 180,E1 9552.481,E2 9552.481} C_VEL
LIN {X 0,Y 185.94,Z 767.546,A -85,B 0,C 180,E1 9548.336,E2 9548.336} C_VEL
LIN {X 0,Y 183.109,Z 765.451,A -85,B 0,C 180,E1 9544.069,E2 9544.069} C_VEL
LIN {X 0,Y 181.035,Z 761.18,A -85,B 0,C 180,E1 9539.366,E2 9539.366} C_VEL
LIN {X 0,Y 179.954,Z 755.203,A -85,B 0,C 180,E1 9534.899,E2 9534.899} C_VEL
LIN {X 0,Y 179.642,Z 748.812,A -85,B 0,C 180,E1 9531.194,E2 9531.194} C_VEL
LIN {X 0,Y 180.777,Z 748.289,A -85,B 0,C 180,E1 9528.837,E2 9528.837} C_VEL
LIN {X 0,Y 181.982,Z 747.58,A -85,B 0,C 180,E1 9527.626,E2 9527.626} C_VEL
LIN {X 0,Y 183.603,Z 746.957,A -85,B 0,C 180,E1 9525.491,E2 9525.491} C_VEL
LIN {X 0,Y 185.294,Z 746.164,A -85,B 0,C 180,E1 9524.025,E2 9524.025} C_VEL
LIN {X 0,Y 188.068,Z 745.062,A -85,B 0,C 180,E1 9521.718,E2 9521.718} C_VEL
LIN {X 0,Y 193.164,Z 743.093,A -85,B 0,C 180,E1 9518.437,E2 9518.437} C_VEL
LIN {X 0,Y 198.883,Z 740.908,A -85,B 0,C 180,E1 9515.5,E2 9515.5} C_VEL
LIN {X 0,Y 205.409,Z 738.39,A -85,B 0,C 180,E1 9512.769,E2 9512.769} C_VEL
LIN {X 0,Y 214.546,Z 734.641,A -85,B 0,C 180,E1 9509.779,E2 9509.779} C_VEL
LIN {X 0,Y 223.957,Z 730.543,A -85,B 0,C 180,E1 9507.301,E2 9507.301} C_VEL
LIN {X 0,Y 234.359,Z 725.793,A -85,B 0,C 180,E1 9505.063,E2 9505.063} C_VEL
LIN {X 0,Y 224.359,Z 740.499,A -85,B 0,C 180,E1 9501.661,E2 9501.661} C_VEL
LIN {X 0,Y 214.666,Z 753.478,A -85,B 0,C 180,E1 9497.782,E2 9497.782} C_VEL
LIN {X 0,Y 205.464,Z 764.929,A -85,B 0,C 180,E1 9493.327,E2 9493.327} C_VEL
LIN {X 0,Y 197.061,Z 774.858,A -85,B 0,C 180,E1 9488.244,E2 9488.244} C_VEL
LIN {X 0,Y 189.8,Z 783.171,A -85,B 0,C 180,E1 9482.503,E2 9482.503} C_VEL
LIN {X 0,Y 184.258,Z 789.536,A -85,B 0,C 180,E1 9476.421,E2 9476.421} C_VEL
LIN {X 0,Y 180.425,Z 794.135,A -85,B 0,C 180,E1 9470.096,E2 9470.096} C_VEL
LIN {X 0,Y 178.201,Z 797.067,A -85,B 0,C 180,E1 9463.631,E2 9463.631} C_VEL
LIN {X 0,Y 177.255,Z 798.406,A -85,B 0,C 180,E1 9457.455,E2 9457.455} C_VEL
LIN {X 0,Y 177.072,Z 798.35,A -85,B 0,C 180,E1 9451.294,E2 9451.294} C_VEL
LIN {X 0,Y 177.538,Z 796.91,A -85,B 0,C 180,E1 9445.154,E2 9445.154} C_VEL
LIN {X 0,Y 179.028,Z 793.913,A -85,B 0,C 180,E1 9438.728,E2 9438.728} C_VEL
LIN {X 0,Y 181.899,Z 789.296,A -85,B 0,C 180,E1 9432.403,E2 9432.403} C_VEL
LIN {X 0,Y 186.363,Z 782.964,A -85,B 0,C 180,E1 9426.273,E2 9426.273} C_VEL
LIN {X 0,Y 192.472,Z 774.773,A -85,B 0,C 180,E1 9420.428,E2 9420.428} C_VEL
LIN {X 0,Y 199.843,Z 764.875,A -85,B 0,C 180,E1 9415.14,E2 9415.14} C_VEL
LIN {X 0,Y 207.878,Z 753.782,A -85,B 0,C 180,E1 9410.587,E2 9410.587} C_VEL
LIN {X 0,Y 216.568,Z 741.098,A -85,B 0,C 180,E1 9406.535,E2 9406.535} C_VEL
LIN {X 0,Y 225.565,Z 726.911,A -85,B 0,C 180,E1 9402.996,E2 9402.996} C_VEL
LIN {X 0,Y 234.318,Z 711.697,A -85,B 0,C 180,E1 9400.009,E2 9400.009} C_VEL
LIN {X 0,Y 242.594,Z 695.586,A -85,B 0,C 180,E1 9397.496,E2 9397.496} C_VEL
LIN {X 0,Y 250.227,Z 678.647,A -85,B 0,C 180,E1 9395.398,E2 9395.398} C_VEL
LIN {X 0,Y 257.055,Z 660.945,A -85,B 0,C 180,E1 9393.655,E2 9393.655} C_VEL
LIN {X 0,Y 258.249,Z 657.293,A -85,B 0,C 180,E1 9393.32,E2 9393.32} C_VEL
LIN {X 0,Y 251.114,Z 666.652,A -85,B 0,C 180,E1 9392.517,E2 9392.517} C_VEL
LIN {X 0,Y 244.721,Z 673.711,A -85,B 0,C 180,E1 9391.533,E2 9391.533} C_VEL
LIN {X 0,Y 243.923,Z 674.509,A -85,B 0,C 180,E1 9391.39,E2 9391.39} C_VEL
LIN {X 0,Y 241.151,Z 677.853,A -85,B 0,C 180,E1 9391.052,E2 9391.052} C_VEL
LIN {X 0,Y 236.803,Z 684.343,A -85,B 0,C 180,E1 9391.054,E2 9391.054} C_VEL
LIN {X 0,Y 232.846,Z 689.969,A -85,B 0,C 180,E1 9391.028,E2 9391.028} C_VEL
LIN {X 0,Y 229.975,Z 693.007,A -85,B 0,C 180,E1 9390.708,E2 9390.708} C_VEL
LIN {X 0,Y 229.497,Z 693.42,A -85,B 0,C 180,E1 9390.617,E2 9390.617} C_VEL
LIN {X 0,Y 223.812,Z 698.215,A -85,B 0,C 180,E1 9389.408,E2 9389.408} C_VEL
LIN {X 0,Y 217.128,Z 703.879,A -85,B 0,C 180,E1 9388.016,E2 9388.016} C_VEL
LIN {X 0,Y 210.587,Z 708.935,A -85,B 0,C 180,E1 9386.205,E2 9386.205} C_VEL
LIN {X 0,Y 204.025,Z 714.039,A -85,B 0,C 180,E1 9384.31,E2 9384.31} C_VEL
LIN {X 0,Y 199.188,Z 717.556,A -85,B 0,C 180,E1 9382.538,E2 9382.538} C_VEL
LIN {X 0,Y 193.474,Z 721.907,A -85,B 0,C 180,E1 9380.259,E2 9380.259} C_VEL
LIN {X 0,Y 190.839,Z 723.759,A -85,B 0,C 180,E1 9378.957,E2 9378.957} C_VEL
LIN {X 0,Y 186.48,Z 727.079,A -85,B 0,C 180,E1 9376.831,E2 9376.831} C_VEL
LIN {X 0,Y 183.922,Z 728.984,A -85,B 0,C 180,E1 9375.127,E2 9375.127} C_VEL
LIN {X 0,Y 180.334,Z 732.018,A -85,B 0,C 180,E1 9372.815,E2 9372.815} C_VEL
LIN {X 0,Y 178.384,Z 733.687,A -85,B 0,C 180,E1 9370.987,E2 9370.987} C_VEL
LIN {X 0,Y 175.523,Z 736.404,A -85,B 0,C 180,E1 9368.519,E2 9368.519} C_VEL
LIN {X 0,Y 174.516,Z 737.46,A -85,B 0,C 180,E1 9366.912,E2 9366.912} C_VEL
LIN {X 0,Y 172.184,Z 740.144,A -85,B 0,C 180,E1 9364.331,E2 9364.331} C_VEL
LIN {X 0,Y 171.58,Z 741.275,A -85,B 0,C 180,E1 9362.339,E2 9362.339} C_VEL
LIN {X 0,Y 171.696,Z 750.343,A -85,B 0,C 180,E1 9357.999,E2 9357.999} C_VEL
LIN {X 0,Y 172.717,Z 759.128,A -85,B 0,C 180,E1 9352.684,E2 9352.684} C_VEL
LIN {X 0,Y 174.825,Z 765.639,A -85,B 0,C 180,E1 9347.449,E2 9347.449} C_VEL
LIN {X 0,Y 177.923,Z 769.965,A -85,B 0,C 180,E1 9342.673,E2 9342.673} C_VEL
LIN {X 0,Y 182.759,Z 772.858,A -85,B 0,C 180,E1 9337.484,E2 9337.484} C_VEL
LIN {X 0,Y 188.59,Z 773.692,A -85,B 0,C 180,E1 9332.875,E2 9332.875} C_VEL
LIN {X 0,Y 196.097,Z 772.729,A -85,B 0,C 180,E1 9328.321,E2 9328.321} C_VEL
LIN {X 0,Y 205.506,Z 769.538,A -85,B 0,C 180,E1 9323.867,E2 9323.867} C_VEL
LIN {X 0,Y 208.792,Z 768.062,A -85,B 0,C 180,E1 9322.481,E2 9322.481} C_VEL
LIN {X 0,Y 204.672,Z 770.934,A -85,B 0,C 180,E1 9320.964,E2 9320.964} C_VEL
LIN {X 0,Y 195.611,Z 783.714,A -85,B 0,C 180,E1 9316.538,E2 9316.538} C_VEL
LIN {X 0,Y 187.332,Z 795.072,A -85,B 0,C 180,E1 9311.44,E2 9311.44} C_VEL
LIN {X 0,Y 180.176,Z 805.018,A -85,B 0,C 180,E1 9305.639,E2 9305.639} C_VEL
LIN {X 0,Y 174.524,Z 813.438,A -85,B 0,C 180,E1 9299.142,E2 9299.142} C_VEL
LIN {X 0,Y 170.834,Z 819.952,A -85,B 0,C 180,E1 9292.361,E2 9292.361} C_VEL
LIN {X 0,Y 168.932,Z 824.963,A -85,B 0,C 180,E1 9285.095,E2 9285.095} C_VEL
LIN {X 0,Y 168.615,Z 827.927,A -85,B 0,C 180,E1 9278.525,E2 9278.525} C_VEL
LIN {X 0,Y 168.857,Z 829.256,A -85,B 0,C 180,E1 9273.055,E2 9273.055} C_VEL
LIN {X 0,Y 168.889,Z 829.578,A -85,B 0,C 180,E1 9268.304,E2 9268.304} C_VEL
LIN {X 0,Y 168.627,Z 828.907,A -85,B 0,C 180,E1 9262.847,E2 9262.847} C_VEL
LIN {X 0,Y 168.726,Z 826.802,A -85,B 0,C 180,E1 9256.288,E2 9256.288} C_VEL
LIN {X 0,Y 170.322,Z 822.784,A -85,B 0,C 180,E1 9248.967,E2 9248.967} C_VEL
LIN {X 0,Y 174.115,Z 816.706,A -85,B 0,C 180,E1 9241.534,E2 9241.534} C_VEL
LIN {X 0,Y 179.988,Z 808.972,A -85,B 0,C 180,E1 9234.708,E2 9234.708} C_VEL
LIN {X 0,Y 187.58,Z 799.602,A -85,B 0,C 180,E1 9228.626,E2 9228.626} C_VEL
LIN {X 0,Y 196.986,Z 788.094,A -85,B 0,C 180,E1 9223.036,E2 9223.036} C_VEL
LIN {X 0,Y 206.866,Z 775.642,A -85,B 0,C 180,E1 9218.463,E2 9218.463} C_VEL
LIN {X 0,Y 217.584,Z 761.141,A -85,B 0,C 180,E1 9214.416,E2 9214.416} C_VEL
LIN {X 0,Y 224.541,Z 750.899,A -85,B 0,C 180,E1 9212.089,E2 9212.089} C_VEL
LIN {X 0,Y 212.452,Z 754.746,A -85,B 0,C 180,E1 9209.613,E2 9209.613} C_VEL
LIN {X 0,Y 205.357,Z 756.569,A -85,B 0,C 180,E1 9207.708,E2 9207.708} C_VEL
LIN {X 0,Y 198.026,Z 762.793,A -85,B 0,C 180,E1 9204.14,E2 9204.14} C_VEL
LIN {X 0,Y 191.252,Z 767.063,A -85,B 0,C 180,E1 9200.183,E2 9200.183} C_VEL
LIN {X 0,Y 185.752,Z 769.214,A -85,B 0,C 180,E1 9196.253,E2 9196.253} C_VEL
LIN {X 0,Y 181.126,Z 769.707,A -85,B 0,C 180,E1 9192.108,E2 9192.108} C_VEL
LIN {X 0,Y 177.179,Z 768.305,A -85,B 0,C 180,E1 9187.456,E2 9187.456} C_VEL
LIN {X 0,Y 174.315,Z 764.904,A -85,B 0,C 180,E1 9182.629,E2 9182.629} C_VEL
LIN {X 0,Y 172.605,Z 759.829,A -85,B 0,C 180,E1 9178.007,E2 9178.007} C_VEL
LIN {X 0,Y 171.925,Z 755.19,A -85,B 0,C 180,E1 9174.66,E2 9174.66} C_VEL
LIN {X 0,Y 172.66,Z 754.632,A -85,B 0,C 180,E1 9172.01,E2 9172.01} C_VEL
LIN {X 0,Y 173.683,Z 753.973,A -85,B 0,C 180,E1 9170.388,E2 9170.388} C_VEL
LIN {X 0,Y 175.276,Z 753.191,A -85,B 0,C 180,E1 9167.814,E2 9167.814} C_VEL
LIN {X 0,Y 176.558,Z 752.611,A -85,B 0,C 180,E1 9166.239,E2 9166.239} C_VEL
LIN {X 0,Y 182.612,Z 750.202,A -85,B 0,C 180,E1 9160.82,E2 9160.82} C_VEL
LIN {X 0,Y 188.422,Z 748.072,A -85,B 0,C 180,E1 9157.208,E2 9157.208} C_VEL
LIN {X 0,Y 194.092,Z 746.05,A -85,B 0,C 180,E1 9154.358,E2 9154.358} C_VEL
LIN {X 0,Y 201.827,Z 743.21,A -85,B 0,C 180,E1 9151.278,E2 9151.278} C_VEL
LIN {X 0,Y 211.292,Z 739.513,A -85,B 0,C 180,E1 9148.313,E2 9148.313} C_VEL
LIN {X 0,Y 221.062,Z 735.505,A -85,B 0,C 180,E1 9145.865,E2 9145.865} C_VEL
LIN {X 0,Y 224.657,Z 733.98,A -85,B 0,C 180,E1 9145.088,E2 9145.088} C_VEL
LIN {X 0,Y 214.548,Z 747.573,A -85,B 0,C 180,E1 9141.531,E2 9141.531} C_VEL
LIN {X 0,Y 204.322,Z 760.153,A -85,B 0,C 180,E1 9137.226,E2 9137.226} C_VEL
LIN {X 0,Y 195.038,Z 770.789,A -85,B 0,C 180,E1 9132.419,E2 9132.419} C_VEL
LIN {X 0,Y 186.642,Z 779.957,A -85,B 0,C 180,E1 9126.87,E2 9126.87} C_VEL
LIN {X 0,Y 179.767,Z 787.275,A -85,B 0,C 180,E1 9120.778,E2 9120.778} C_VEL
LIN {X 0,Y 174.701,Z 792.746,A -85,B 0,C 180,E1 9114.336,E2 9114.336} C_VEL
LIN {X 0,Y 171.406,Z 796.506,A -85,B 0,C 180,E1 9107.658,E2 9107.658} C_VEL
LIN {X 0,Y 169.69,Z 798.647,A -85,B 0,C 180,E1 9100.869,E2 9100.869} C_VEL
LIN {X 0,Y 169.117,Z 799.27,A -85,B 0,C 180,E1 9094.408,E2 9094.408} C_VEL
LIN {X 0,Y 169.243,Z 798.56,A -85,B 0,C 180,E1 9088.307,E2 9088.307} C_VEL
LIN {X 0,Y 170.158,Z 796.499,A -85,B 0,C 180,E1 9081.893,E2 9081.893} C_VEL
LIN {X 0,Y 172.393,Z 792.816,A -85,B 0,C 180,E1 9075.215,E2 9075.215} C_VEL
LIN {X 0,Y 176.234,Z 787.475,A -85,B 0,C 180,E1 9068.709,E2 9068.709} C_VEL
LIN {X 0,Y 181.775,Z 780.362,A -85,B 0,C 180,E1 9062.481,E2 9062.481} C_VEL
LIN {X 0,Y 189.016,Z 771.31,A -85,B 0,C 180,E1 9056.623,E2 9056.623} C_VEL
LIN {X 0,Y 197.364,Z 760.615,A -85,B 0,C 180,E1 9051.455,E2 9051.455} C_VEL
LIN {X 0,Y 206.132,Z 748.828,A -85,B 0,C 180,E1 9047.093,E2 9047.093} C_VEL
LIN {X 0,Y 214.87,Z 736.255,A -85,B 0,C 180,E1 9043.454,E2 9043.454} C_VEL
LIN {X 0,Y 223.917,Z 722.054,A -85,B 0,C 180,E1 9040.22,E2 9040.22} C_VEL
LIN {X 0,Y 232.886,Z 706.424,A -85,B 0,C 180,E1 9037.413,E2 9037.413} C_VEL
LIN {X 0,Y 241.607,Z 689.165,A -85,B 0,C 180,E1 9034.975,E2 9034.975} C_VEL
LIN {X 0,Y 247.39,Z 675.967,A -85,B 0,C 180,E1 9033.428,E2 9033.428} C_VEL
LIN {X 0,Y 241.133,Z 682.19,A -85,B 0,C 180,E1 9032.479,E2 9032.479} C_VEL
LIN {X 0,Y 233.05,Z 690.296,A -85,B 0,C 180,E1 9031.275,E2 9031.275} C_VEL
LIN {X 0,Y 229.497,Z 693.42,A -85,B 0,C 180,E1 9030.617,E2 9030.617} C_VEL
LIN {X 0,Y 226.499,Z 696.406,A -85,B 0,C 180,E1 9030.182,E2 9030.182} C_VEL
LIN {X 0,Y 217.01,Z 707.274,A -85,B 0,C 180,E1 9029.702,E2 9029.702} C_VEL
LIN {X 0,Y 213.943,Z 709.971,A -85,B 0,C 180,E1 9029.247,E2 9029.247} C_VEL
LIN {X 0,Y 213.454,Z 710.326,A -85,B 0,C 180,E1 9029.134,E2 9029.134} C_VEL
LIN {X 0,Y 207.691,Z 714.49,A -85,B 0,C 180,E1 9027.648,E2 9027.648} C_VEL
LIN {X 0,Y 200.746,Z 719.551,A -85,B 0,C 180,E1 9025.68,E2 9025.68} C_VEL
LIN {X 0,Y 196.004,Z 722.75,A -85,B 0,C 180,E1 9024.06,E2 9024.06} C_VEL
LIN {X 0,Y 189.676,Z 727.18,A -85,B 0,C 180,E1 9021.655,E2 9021.655} C_VEL
LIN {X 0,Y 186.875,Z 729.092,A -85,B 0,C 180,E1 9020.353,E2 9020.353} C_VEL
LIN {X 0,Y 181.736,Z 732.678,A -85,B 0,C 180,E1 9017.862,E2 9017.862} C_VEL
LIN {X 0,Y 179.009,Z 734.585,A -85,B 0,C 180,E1 9016.218,E2 9016.218} C_VEL
LIN {X 0,Y 174.974,Z 737.642,A -85,B 0,C 180,E1 9013.551,E2 9013.551} C_VEL
LIN {X 0,Y 173.143,Z 739.099,A -85,B 0,C 180,E1 9012,E2 9012} C_VEL
LIN {X 0,Y 169.976,Z 741.917,A -85,B 0,C 180,E1 9009.14,E2 9009.14} C_VEL
LIN {X 0,Y 169.027,Z 742.823,A -85,B 0,C 180,E1 9007.821,E2 9007.821} C_VEL
LIN {X 0,Y 166.404,Z 745.544,A -85,B 0,C 180,E1 9004.827,E2 9004.827} C_VEL
LIN {X 0,Y 165.461,Z 746.867,A -85,B 0,C 180,E1 9002.772,E2 9002.772} C_VEL
LIN {X 0,Y 163.824,Z 749.4,A -85,B 0,C 180,E1 8999.652,E2 8999.652} C_VEL
LIN {X 0,Y 163.719,Z 750.525,A -85,B 0,C 180,E1 8997.726,E2 8997.726} C_VEL
LIN {X 0,Y 164.682,Z 758.887,A -85,B 0,C 180,E1 8992.676,E2 8992.676} C_VEL
LIN {X 0,Y 166.858,Z 766,A -85,B 0,C 180,E1 8987.191,E2 8987.191} C_VEL
LIN {X 0,Y 170.606,Z 771.302,A -85,B 0,C 180,E1 8981.551,E2 8981.551} C_VEL
LIN {X 0,Y 175.506,Z 774.382,A -85,B 0,C 180,E1 8976.499,E2 8976.499} C_VEL
LIN {X 0,Y 182.154,Z 775.743,A -85,B 0,C 180,E1 8971.476,E2 8971.476} C_VEL
LIN {X 0,Y 190.181,Z 775.147,A -85,B 0,C 180,E1 8966.855,E2 8966.855} C_VEL
LIN {X 0,Y 199.493,Z 772.737,A -85,B 0,C 180,E1 8962.668,E2 8962.668} C_VEL
LIN {X 0,Y 195.416,Z 775.38,A -85,B 0,C 180,E1 8961.052,E2 8961.052} C_VEL
LIN {X 0,Y 185.844,Z 787.998,A -85,B 0,C 180,E1 8956.132,E2 8956.132} C_VEL
LIN {X 0,Y 177.176,Z 799.175,A -85,B 0,C 180,E1 8950.374,E2 8950.374} C_VEL
LIN {X 0,Y 170.107,Z 808.592,A -85,B 0,C 180,E1 8943.945,E2 8943.945} C_VEL
LIN {X 0,Y 165.002,Z 816.067,A -85,B 0,C 180,E1 8937.031,E2 8937.031} C_VEL
LIN {X 0,Y 161.824,Z 822.001,A -85,B 0,C 180,E1 8929.49,E2 8929.49} C_VEL
LIN {X 0,Y 160.679,Z 825.944,A -85,B 0,C 180,E1 8922.214,E2 8922.214} C_VEL
LIN {X 0,Y 160.76,Z 828.084,A -85,B 0,C 180,E1 8915.667,E2 8915.667} C_VEL
LIN {X 0,Y 160.962,Z 828.809,A -85,B 0,C 180,E1 8910.356,E2 8910.356} C_VEL
LIN {X 0,Y 160.762,Z 828.628,A -85,B 0,C 180,E1 8905.005,E2 8905.005} C_VEL
LIN {X 0,Y 160.599,Z 827.159,A -85,B 0,C 180,E1 8898.508,E2 8898.508} C_VEL
LIN {X 0,Y 161.611,Z 823.994,A -85,B 0,C 180,E1 8891.185,E2 8891.185} C_VEL
LIN {X 0,Y 164.821,Z 818.714,A -85,B 0,C 180,E1 8883.326,E2 8883.326} C_VEL
LIN {X 0,Y 170.213,Z 811.794,A -85,B 0,C 180,E1 8876.079,E2 8876.079} C_VEL
LIN {X 0,Y 177.476,Z 803.315,A -85,B 0,C 180,E1 8869.617,E2 8869.617} C_VEL
LIN {X 0,Y 186.668,Z 792.784,A -85,B 0,C 180,E1 8863.688,E2 8863.688} C_VEL
LIN {X 0,Y 196.997,Z 780.672,A -85,B 0,C 180,E1 8858.59,E2 8858.59} C_VEL
LIN {X 0,Y 207.406,Z 767.708,A -85,B 0,C 180,E1 8854.476,E2 8854.476} C_VEL
LIN {X 0,Y 214.376,Z 758.427,A -85,B 0,C 180,E1 8852.119,E2 8852.119} C_VEL
LIN {X 0,Y 202.271,Z 761.478,A -85,B 0,C 180,E1 8849.298,E2 8849.298} C_VEL
LIN {X 0,Y 196.219,Z 762.766,A -85,B 0,C 180,E1 8847.461,E2 8847.461} C_VEL
LIN {X 0,Y 188.763,Z 767.529,A -85,B 0,C 180,E1 8843.737,E2 8843.737} C_VEL
LIN {X 0,Y 182.357,Z 770.333,A -85,B 0,C 180,E1 8839.872,E2 8839.872} C_VEL
LIN {X 0,Y 176.464,Z 771.504,A -85,B 0,C 180,E1 8835.443,E2 8835.443} C_VEL
LIN {X 0,Y 171.64,Z 770.728,A -85,B 0,C 180,E1 8830.742,E2 8830.742} C_VEL
LIN {X 0,Y 167.958,Z 767.999,A -85,B 0,C 180,E1 8825.807,E2 8825.807} C_VEL
LIN {X 0,Y 165.573,Z 763.62,A -85,B 0,C 180,E1 8821.037,E2 8821.037} C_VEL
LIN {X 0,Y 164.862,Z 761.356,A -85,B 0,C 180,E1 8818.956,E2 8818.956} C_VEL
LIN {X 0,Y 165.142,Z 760.612,A -85,B 0,C 180,E1 8815.484,E2 8815.484} C_VEL
LIN {X 0,Y 165.689,Z 760.093,A -85,B 0,C 180,E1 8813.763,E2 8813.763} C_VEL
LIN {X 0,Y 167.055,Z 759.193,A -85,B 0,C 180,E1 8810.699,E2 8810.699} C_VEL
LIN {X 0,Y 169.704,Z 757.909,A -85,B 0,C 180,E1 8806.715,E2 8806.715} C_VEL
LIN {X 0,Y 172.971,Z 756.614,A -85,B 0,C 180,E1 8803.199,E2 8803.199} C_VEL
LIN {X 0,Y 177.539,Z 754.965,A -85,B 0,C 180,E1 8799.562,E2 8799.562} C_VEL
LIN {X 0,Y 183.065,Z 753.085,A -85,B 0,C 180,E1 8796.159,E2 8796.159} C_VEL
LIN {X 0,Y 190.171,Z 750.637,A -85,B 0,C 180,E1 8792.778,E2 8792.778} C_VEL
LIN {X 0,Y 197.609,Z 748.079,A -85,B 0,C 180,E1 8789.909,E2 8789.909} C_VEL
LIN {X 0,Y 207.812,Z 744.337,A -85,B 0,C 180,E1 8786.844,E2 8786.844} C_VEL
LIN {X 0,Y 214.671,Z 741.868,A -85,B 0,C 180,E1 8785.047,E2 8785.047} C_VEL
LIN {X 0,Y 204.115,Z 754.82,A -85,B 0,C 180,E1 8781.157,E2 8781.157} C_VEL
LIN {X 0,Y 193.953,Z 766.278,A -85,B 0,C 180,E1 8776.626,E2 8776.626} C_VEL
LIN {X 0,Y 184.542,Z 776.204,A -85,B 0,C 180,E1 8771.377,E2 8771.377} C_VEL
LIN {X 0,Y 176.28,Z 784.548,A -85,B 0,C 180,E1 8765.349,E2 8765.349} C_VEL
LIN {X 0,Y 169.843,Z 790.923,A -85,B 0,C 180,E1 8758.864,E2 8758.864} C_VEL
LIN {X 0,Y 165.287,Z 795.534,A -85,B 0,C 180,E1 8752.028,E2 8752.028} C_VEL
LIN {X 0,Y 162.567,Z 798.48,A -85,B 0,C 180,E1 8744.971,E2 8744.971} C_VEL
LIN {X 0,Y 161.385,Z 799.835,A -85,B 0,C 180,E1 8738.193,E2 8738.193} C_VEL
LIN {X 0,Y 161.126,Z 799.813,A -85,B 0,C 180,E1 8731.778,E2 8731.778} C_VEL
LIN {X 0,Y 161.563,Z 798.591,A -85,B 0,C 180,E1 8725.386,E2 8725.386} C_VEL
LIN {X 0,Y 163.157,Z 795.806,A -85,B 0,C 180,E1 8718.333,E2 8718.333} C_VEL
LIN {X 0,Y 166.312,Z 791.423,A -85,B 0,C 180,E1 8711.42,E2 8711.42} C_VEL
LIN {X 0,Y 171.242,Z 785.332,A -85,B 0,C 180,E1 8704.771,E2 8704.771} C_VEL
LIN {X 0,Y 177.584,Z 777.832,A -85,B 0,C 180,E1 8698.802,E2 8698.802} C_VEL
LIN {X 0,Y 185.467,Z 768.502,A -85,B 0,C 180,E1 8693.244,E2 8693.244} C_VEL
LIN {X 0,Y 194.244,Z 757.744,A -85,B 0,C 180,E1 8688.393,E2 8688.393} C_VEL
LIN {X 0,Y 203.574,Z 745.585,A -85,B 0,C 180,E1 8684.186,E2 8684.186} C_VEL
LIN {X 0,Y 213.177,Z 731.987,A -85,B 0,C 180,E1 8680.551,E2 8680.551} C_VEL
LIN {X 0,Y 222.811,Z 716.865,A -85,B 0,C 180,E1 8677.412,E2 8677.412} C_VEL
LIN {X 0,Y 231.926,Z 700.742,A -85,B 0,C 180,E1 8674.788,E2 8674.788} C_VEL
LIN {X 0,Y 236.75,Z 691.206,A -85,B 0,C 180,E1 8673.488,E2 8673.488} C_VEL
LIN {X 0,Y 227.969,Z 698.86,A -85,B 0,C 180,E1 8672.054,E2 8672.054} C_VEL
LIN {X 0,Y 222.871,Z 702.885,A -85,B 0,C 180,E1 8671.06,E2 8671.06} C_VEL
LIN {X 0,Y 215.089,Z 709.156,A -85,B 0,C 180,E1 8669.523,E2 8669.523} C_VEL
LIN {X 0,Y 213.454,Z 710.326,A -85,B 0,C 180,E1 8669.134,E2 8669.134} C_VEL
LIN {X 0,Y 209.802,Z 713.446,A -85,B 0,C 180,E1 8668.504,E2 8668.504} C_VEL
LIN {X 0,Y 200.655,Z 722.3,A -85,B 0,C 180,E1 8667.709,E2 8667.709} C_VEL
LIN {X 0,Y 197.097,Z 725.091,A -85,B 0,C 180,E1 8666.999,E2 8666.999} C_VEL
LIN {X 0,Y 196.64,Z 725.385,A -85,B 0,C 180,E1 8666.854,E2 8666.854} C_VEL
LIN {X 0,Y 186.459,Z 731.934,A -85,B 0,C 180,E1 8663.38,E2 8663.38} C_VEL
LIN {X 0,Y 182.225,Z 734.639,A -85,B 0,C 180,E1 8661.571,E2 8661.571} C_VEL
LIN {X 0,Y 176.677,Z 738.245,A -85,B 0,C 180,E1 8658.82,E2 8658.82} C_VEL
LIN {X 0,Y 170.273,Z 742.566,A -85,B 0,C 180,E1 8654.975,E2 8654.975} C_VEL
LIN {X 0,Y 168.324,Z 743.949,A -85,B 0,C 180,E1 8653.396,E2 8653.396} C_VEL
LIN {X 0,Y 164.595,Z 746.929,A -85,B 0,C 180,E1 8650.23,E2 8650.23} C_VEL
LIN {X 0,Y 163.048,Z 748.292,A -85,B 0,C 180,E1 8648.465,E2 8648.465} C_VEL
LIN {X 0,Y 160.524,Z 750.793,A -85,B 0,C 180,E1 8645.362,E2 8645.362} C_VEL
LIN {X 0,Y 159.616,Z 751.898,A -85,B 0,C 180,E1 8643.593,E2 8643.593} C_VEL
LIN {X 0,Y 157.74,Z 754.531,A -85,B 0,C 180,E1 8640.001,E2 8640.001} C_VEL
LIN {X 0,Y 157.424,Z 755.534,A -85,B 0,C 180,E1 8638.181,E2 8638.181} C_VEL
LIN {X 0,Y 156.495,Z 758.391,A -85,B 0,C 180,E1 8634.134,E2 8634.134} C_VEL
LIN {X 0,Y 156.854,Z 759.564,A -85,B 0,C 180,E1 8631.94,E2 8631.94} C_VEL
LIN {X 0,Y 159.256,Z 766.912,A -85,B 0,C 180,E1 8626.199,E2 8626.199} C_VEL
LIN {X 0,Y 163.069,Z 772.288,A -85,B 0,C 180,E1 8620.666,E2 8620.666} C_VEL
LIN {X 0,Y 168.67,Z 775.998,A -85,B 0,C 180,E1 8615.111,E2 8615.111} C_VEL
LIN {X 0,Y 175.816,Z 777.693,A -85,B 0,C 180,E1 8609.971,E2 8609.971} C_VEL
LIN {X 0,Y 184.404,Z 777.581,A -85,B 0,C 180,E1 8605.298,E2 8605.298} C_VEL
LIN {X 0,Y 189.884,Z 776.73,A -85,B 0,C 180,E1 8602.733,E2 8602.733} C_VEL
LIN {X 0,Y 186.726,Z 778.771,A -85,B 0,C 180,E1 8601.425,E2 8601.425} C_VEL
LIN {X 0,Y 177.055,Z 790.764,A -85,B 0,C 180,E1 8596.29,E2 8596.29} C_VEL
LIN {X 0,Y 168.435,Z 801.194,A -85,B 0,C 180,E1 8590.319,E2 8590.319} C_VEL
LIN {X 0,Y 161.33,Z 810.114,A -85,B 0,C 180,E1 8583.476,E2 8583.476} C_VEL
LIN {X 0,Y 156.382,Z 817.145,A -85,B 0,C 180,E1 8576.178,E2 8576.178} C_VEL
LIN {X 0,Y 153.485,Z 822.562,A -85,B 0,C 180,E1 8568.221,E2 8568.221} C_VEL
LIN {X 0,Y 152.647,Z 826.026,A -85,B 0,C 180,E1 8560.568,E2 8560.568} C_VEL
LIN {X 0,Y 152.866,Z 827.688,A -85,B 0,C 180,E1 8554.126,E2 8554.126} C_VEL
LIN {X 0,Y 152.971,Z 828.143,A -85,B 0,C 180,E1 8548.876,E2 8548.876} C_VEL
LIN {X 0,Y 152.696,Z 827.666,A -85,B 0,C 180,E1 8543.231,E2 8543.231} C_VEL
LIN {X 0,Y 152.775,Z 825.773,A -85,B 0,C 180,E1 8535.986,E2 8535.986} C_VEL
LIN {X 0,Y 154.562,Z 822.038,A -85,B 0,C 180,E1 8527.963,E2 8527.963} C_VEL
LIN {X 0,Y 158.632,Z 816.532,A -85,B 0,C 180,E1 8520.136,E2 8520.136} C_VEL
LIN {X 0,Y 165.123,Z 809.087,A -85,B 0,C 180,E1 8512.733,E2 8512.733} C_VEL
LIN {X 0,Y 173.934,Z 799.629,A -85,B 0,C 180,E1 8505.927,E2 8505.927} C_VEL
LIN {X 0,Y 183.71,Z 789.062,A -85,B 0,C 180,E1 8500.362,E2 8500.362} C_VEL
LIN {X 0,Y 194.373,Z 777.001,A -85,B 0,C 180,E1 8495.633,E2 8495.633} C_VEL
LIN {X 0,Y 204.004,Z 765.264,A -85,B 0,C 180,E1 8492.057,E2 8492.057} C_VEL
LIN {X 0,Y 192.894,Z 767.448,A -85,B 0,C 180,E1 8489.159,E2 8489.159} C_VEL
LIN {X 0,Y 185.651,Z 768.72,A -85,B 0,C 180,E1 8486.615,E2 8486.615} C_VEL
LIN {X 0,Y 177.912,Z 771.971,A -85,B 0,C 180,E1 8482.466,E2 8482.466} C_VEL
LIN {X 0,Y 171.265,Z 773.247,A -85,B 0,C 180,E1 8478.023,E2 8478.023} C_VEL
LIN {X 0,Y 166.065,Z 772.776,A -85,B 0,C 180,E1 8473.579,E2 8473.579} C_VEL
LIN {X 0,Y 161.644,Z 770.43,A -85,B 0,C 180,E1 8468.536,E2 8468.536} C_VEL
LIN {X 0,Y 159.015,Z 767.315,A -85,B 0,C 180,E1 8464.326,E2 8464.326} C_VEL
LIN {X 0,Y 158.241,Z 766.476,A -85,B 0,C 180,E1 8459.999,E2 8459.999} C_VEL
LIN {X 0,Y 158.954,Z 765.112,A -85,B 0,C 180,E1 8454.585,E2 8454.585} C_VEL
LIN {X 0,Y 160.878,Z 763.845,A -85,B 0,C 180,E1 8449.977,E2 8449.977} C_VEL
LIN {X 0,Y 163.695,Z 762.581,A -85,B 0,C 180,E1 8445.857,E2 8445.857} C_VEL
LIN {X 0,Y 167.559,Z 761.14,A -85,B 0,C 180,E1 8441.922,E2 8441.922} C_VEL
LIN {X 0,Y 172.023,Z 759.644,A -85,B 0,C 180,E1 8438.433,E2 8438.433} C_VEL
LIN {X 0,Y 182.231,Z 756.431,A -85,B 0,C 180,E1 8432.731,E2 8432.731} C_VEL
LIN {X 0,Y 193.261,Z 752.796,A -85,B 0,C 180,E1 8428.496,E2 8428.496} C_VEL
LIN {X 0,Y 204.239,Z 749.028,A -85,B 0,C 180,E1 8425.332,E2 8425.332} C_VEL
LIN {X 0,Y 204.951,Z 748.831,A -85,B 0,C 180,E1 8425.111,E2 8425.111} C_VEL
LIN {X 0,Y 193.654,Z 761.502,A -85,B 0,C 180,E1 8420.758,E2 8420.758} C_VEL
LIN {X 0,Y 183.569,Z 771.907,A -85,B 0,C 180,E1 8415.97,E2 8415.97} C_VEL
LIN {X 0,Y 174.322,Z 780.875,A -85,B 0,C 180,E1 8410.402,E2 8410.402} C_VEL
LIN {X 0,Y 166.234,Z 788.422,A -85,B 0,C 180,E1 8403.895,E2 8403.895} C_VEL
LIN {X 0,Y 159.964,Z 794.197,A -85,B 0,C 180,E1 8396.639,E2 8396.639} C_VEL
LIN {X 0,Y 155.908,Z 798.043,A -85,B 0,C 180,E1 8389.091,E2 8389.091} C_VEL
LIN {X 0,Y 153.86,Z 800.12,A -85,B 0,C 180,E1 8381.622,E2 8381.622} C_VEL
LIN {X 0,Y 153.194,Z 800.706,A -85,B 0,C 180,E1 8374.867,E2 8374.867} C_VEL
LIN {X 0,Y 153.318,Z 800.023,A -85,B 0,C 180,E1 8368.132,E2 8368.132} C_VEL
LIN {X 0,Y 154.385,Z 798.014,A -85,B 0,C 180,E1 8361.058,E2 8361.058} C_VEL
LIN {X 0,Y 156.995,Z 794.389,A -85,B 0,C 180,E1 8353.726,E2 8353.726} C_VEL
LIN {X 0,Y 161.432,Z 789.113,A -85,B 0,C 180,E1 8346.647,E2 8346.647} C_VEL
LIN {X 0,Y 167.749,Z 782.078,A -85,B 0,C 180,E1 8339.955,E2 8339.955} C_VEL
LIN {X 0,Y 175.887,Z 773.115,A -85,B 0,C 180,E1 8333.757,E2 8333.757} C_VEL
LIN {X 0,Y 185.147,Z 762.511,A -85,B 0,C 180,E1 8328.375,E2 8328.375} C_VEL
LIN {X 0,Y 194.964,Z 750.581,A -85,B 0,C 180,E1 8323.817,E2 8323.817} C_VEL
LIN {X 0,Y 204.892,Z 737.493,A -85,B 0,C 180,E1 8319.99,E2 8319.99} C_VEL
LIN {X 0,Y 215.027,Z 722.755,A -85,B 0,C 180,E1 8316.667,E2 8316.667} C_VEL
LIN {X 0,Y 224.681,Z 707.022,A -85,B 0,C 180,E1 8313.906,E2 8313.906} C_VEL
LIN {X 0,Y 226.16,Z 704.399,A -85,B 0,C 180,E1 8313.473,E2 8313.473} C_VEL
LIN {X 0,Y 220.996,Z 708.311,A -85,B 0,C 180,E1 8312.576,E2 8312.576} C_VEL
LIN {X 0,Y 213.066,Z 714.29,A -85,B 0,C 180,E1 8311.079,E2 8311.079} C_VEL
LIN {X 0,Y 205.006,Z 719.743,A -85,B 0,C 180,E1 8309.188,E2 8309.188} C_VEL
LIN {X 0,Y 197.431,Z 724.884,A -85,B 0,C 180,E1 8307.117,E2 8307.117} C_VEL
LIN {X 0,Y 196.64,Z 725.385,A -85,B 0,C 180,E1 8306.854,E2 8306.854} C_VEL
LIN {X 0,Y 193.141,Z 727.912,A -85,B 0,C 180,E1 8305.992,E2 8305.992} C_VEL
LIN {X 0,Y 182.119,Z 736.96,A -85,B 0,C 180,E1 8304.356,E2 8304.356} C_VEL
LIN {X 0,Y 179.622,Z 738.675,A -85,B 0,C 180,E1 8303.66,E2 8303.66} C_VEL
LIN {X 0,Y 173.399,Z 742.482,A -85,B 0,C 180,E1 8300.948,E2 8300.948} C_VEL
LIN {X 0,Y 169.624,Z 744.797,A -85,B 0,C 180,E1 8298.919,E2 8298.919} C_VEL
LIN {X 0,Y 164.328,Z 748.098,A -85,B 0,C 180,E1 8295.53,E2 8295.53} C_VEL
LIN {X 0,Y 158.998,Z 751.878,A -85,B 0,C 180,E1 8291.243,E2 8291.243} C_VEL
LIN {X 0,Y 157.362,Z 753.185,A -85,B 0,C 180,E1 8289.51,E2 8289.51} C_VEL
LIN {X 0,Y 154.478,Z 755.811,A -85,B 0,C 180,E1 8285.946,E2 8285.946} C_VEL
LIN {X 0,Y 153.105,Z 757.32,A -85,B 0,C 180,E1 8283.746,E2 8283.746} C_VEL
LIN {X 0,Y 151.436,Z 759.663,A -85,B 0,C 180,E1 8280.001,E2 8280.001} C_VEL
LIN {X 0,Y 150.692,Z 761.107,A -85,B 0,C 180,E1 8277.72,E2 8277.72} C_VEL
LIN {X 0,Y 150.198,Z 763.791,A -85,B 0,C 180,E1 8273.119,E2 8273.119} C_VEL
LIN {X 0,Y 151.561,Z 768.208,A -85,B 0,C 180,E1 8265.483,E2 8265.483} C_VEL
LIN {X 0,Y 152.605,Z 769.369,A -85,B 0,C 180,E1 8263.638,E2 8263.638} C_VEL
LIN {X 0,Y 157.474,Z 774.82,A -85,B 0,C 180,E1 8257.608,E2 8257.608} C_VEL
LIN {X 0,Y 163.599,Z 778.175,A -85,B 0,C 180,E1 8252.325,E2 8252.325} C_VEL
LIN {X 0,Y 172.157,Z 779.892,A -85,B 0,C 180,E1 8246.913,E2 8246.913} C_VEL
LIN {X 0,Y 180.322,Z 779.859,A -85,B 0,C 180,E1 8242.886,E2 8242.886} C_VEL
LIN {X 0,Y 178.625,Z 781.229,A -85,B 0,C 180,E1 8242.116,E2 8242.116} C_VEL
LIN {X 0,Y 168.76,Z 792.683,A -85,B 0,C 180,E1 8236.781,E2 8236.781} C_VEL
LIN {X 0,Y 160.007,Z 802.715,A -85,B 0,C 180,E1 8230.533,E2 8230.533} C_VEL
LIN {X 0,Y 152.851,Z 811.167,A -85,B 0,C 180,E1 8223.331,E2 8223.331} C_VEL
LIN {X 0,Y 147.786,Z 818.028,A -85,B 0,C 180,E1 8215.229,E2 8215.229} C_VEL
LIN {X 0,Y 145.265,Z 822.805,A -85,B 0,C 180,E1 8207.216,E2 8207.216} C_VEL
LIN {X 0,Y 144.665,Z 825.795,A -85,B 0,C 180,E1 8199.548,E2 8199.548} C_VEL
LIN {X 0,Y 144.938,Z 827.124,A -85,B 0,C 180,E1 8193.164,E2 8193.164} C_VEL
LIN {X 0,Y 144.969,Z 827.438,A -85,B 0,C 180,E1 8188.024,E2 8188.024} C_VEL
LIN {X 0,Y 144.659,Z 826.821,A -85,B 0,C 180,E1 8182.054,E2 8182.054} C_VEL
LIN {X 0,Y 144.964,Z 824.778,A -85,B 0,C 180,E1 8174.395,E2 8174.395} C_VEL
LIN {X 0,Y 147.259,Z 820.88,A -85,B 0,C 180,E1 8165.959,E2 8165.959} C_VEL
LIN {X 0,Y 152.04,Z 815.156,A -85,B 0,C 180,E1 8157.813,E2 8157.813} C_VEL
LIN {X 0,Y 159.764,Z 807.133,A -85,B 0,C 180,E1 8149.863,E2 8149.863} C_VEL
LIN {X 0,Y 169.038,Z 797.871,A -85,B 0,C 180,E1 8143.318,E2 8143.318} C_VEL
LIN {X 0,Y 179.593,Z 787.037,A -85,B 0,C 180,E1 8137.761,E2 8137.761} C_VEL
LIN {X 0,Y 191.603,Z 774.009,A -85,B 0,C 180,E1 8132.842,E2 8132.842} C_VEL
LIN {X 0,Y 193.85,Z 771.415,A -85,B 0,C 180,E1 8132.011,E2 8132.011} C_VEL
LIN {X 0,Y 181.887,Z 773.094,A -85,B 0,C 180,E1 8128.412,E2 8128.412} C_VEL
LIN {X 0,Y 172.348,Z 774.065,A -85,B 0,C 180,E1 8124.323,E2 8124.323} C_VEL
LIN {X 0,Y 165.15,Z 775.12,A -85,B 0,C 180,E1 8119.817,E2 8119.817} C_VEL
LIN {X 0,Y 159.086,Z 774.308,A -85,B 0,C 180,E1 8114.931,E2 8114.931} C_VEL
LIN {X 0,Y 155.796,Z 773.111,A -85,B 0,C 180,E1 8111.474,E2 8111.474} C_VEL
LIN {X 0,Y 152.633,Z 772.042,A -85,B 0,C 180,E1 8105.261,E2 8105.261} C_VEL
LIN {X 0,Y 151.698,Z 770.822,A -85,B 0,C 180,E1 8099.325,E2 8099.325} C_VEL
LIN {X 0,Y 152.508,Z 769.555,A -85,B 0,C 180,E1 8093.977,E2 8093.977} C_VEL
LIN {X 0,Y 154.328,Z 768.444,A -85,B 0,C 180,E1 8089.547,E2 8089.547} C_VEL
LIN {X 0,Y 160.818,Z 765.949,A -85,B 0,C 180,E1 8081.512,E2 8081.512} C_VEL
LIN {X 0,Y 171.072,Z 762.769,A -85,B 0,C 180,E1 8074.372,E2 8074.372} C_VEL
LIN {X 0,Y 185.475,Z 758.444,A -85,B 0,C 180,E1 8068.108,E2 8068.108} C_VEL
LIN {X 0,Y 195.007,Z 755.509,A -85,B 0,C 180,E1 8065.122,E2 8065.122} C_VEL
LIN {X 0,Y 183.763,Z 767.066,A -85,B 0,C 180,E1 8060.591,E2 8060.591} C_VEL
LIN {X 0,Y 173.048,Z 777.204,A -85,B 0,C 180,E1 8055.176,E2 8055.176} C_VEL
LIN {X 0,Y 163.688,Z 785.523,A -85,B 0,C 180,E1 8048.989,E2 8048.989} C_VEL
LIN {X 0,Y 156.108,Z 792.026,A -85,B 0,C 180,E1 8042.115,E2 8042.115} C_VEL
LIN {X 0,Y 150.368,Z 796.935,A -85,B 0,C 180,E1 8034.347,E2 8034.347} C_VEL
LIN {X 0,Y 146.913,Z 799.985,A -85,B 0,C 180,E1 8026.203,E2 8026.203} C_VEL
LIN {X 0,Y 145.491,Z 801.282,A -85,B 0,C 180,E1 8018.696,E2 8018.696} C_VEL
LIN {X 0,Y 145.193,Z 801.234,A -85,B 0,C 180,E1 8011.579,E2 8011.579} C_VEL
LIN {X 0,Y 145.741,Z 799.978,A -85,B 0,C 180,E1 8004.489,E2 8004.489} C_VEL
LIN {X 0,Y 147.694,Z 797.171,A -85,B 0,C 180,E1 7996.693,E2 7996.693} C_VEL
LIN {X 0,Y 151.48,Z 792.768,A -85,B 0,C 180,E1 7989.119,E2 7989.119} C_VEL
LIN {X 0,Y 157.252,Z 786.666,A -85,B 0,C 180,E1 7981.932,E2 7981.932} C_VEL
LIN {X 0,Y 164.969,Z 778.732,A -85,B 0,C 180,E1 7975.269,E2 7975.269} C_VEL
LIN {X 0,Y 173.951,Z 769.295,A -85,B 0,C 180,E1 7969.495,E2 7969.495} C_VEL
LIN {X 0,Y 183.776,Z 758.378,A -85,B 0,C 180,E1 7964.543,E2 7964.543} C_VEL
LIN {X 0,Y 194.073,Z 746.03,A -85,B 0,C 180,E1 7960.315,E2 7960.315} C_VEL
LIN {X 0,Y 204.554,Z 732.241,A -85,B 0,C 180,E1 7956.713,E2 7956.713} C_VEL
LIN {X 0,Y 214.971,Z 716.959,A -85,B 0,C 180,E1 7953.638,E2 7953.638} C_VEL
LIN {X 0,Y 215.199,Z 716.44,A -85,B 0,C 180,E1 7953.487,E2 7953.487} C_VEL
LIN {X 0,Y 196.273,Z 728.711,A -85,B 0,C 180,E1 7949.279,E2 7949.279} C_VEL
LIN {X 0,Y 189.695,Z 732.733,A -85,B 0,C 180,E1 7947.296,E2 7947.296} C_VEL
LIN {X 0,Y 182.046,Z 737.276,A -85,B 0,C 180,E1 7944.673,E2 7944.673} C_VEL
LIN {X 0,Y 179.622,Z 738.675,A -85,B 0,C 180,E1 7943.66,E2 7943.66} C_VEL
LIN {X 0,Y 172.466,Z 743.618,A -85,B 0,C 180,E1 7941.406,E2 7941.406} C_VEL
LIN {X 0,Y 161.715,Z 751.156,A -85,B 0,C 180,E1 7937.925,E2 7937.925} C_VEL
LIN {X 0,Y 157.57,Z 753.878,A -85,B 0,C 180,E1 7935.822,E2 7935.822} C_VEL
LIN {X 0,Y 153.076,Z 756.815,A -85,B 0,C 180,E1 7932.066,E2 7932.066} C_VEL
LIN {X 0,Y 148.498,Z 760.416,A -85,B 0,C 180,E1 7926.963,E2 7926.963} C_VEL
LIN {X 0,Y 146.726,Z 762.163,A -85,B 0,C 180,E1 7924.3,E2 7924.3} C_VEL
LIN {X 0,Y 144.484,Z 765.347,A -85,B 0,C 180,E1 7918.812,E2 7918.812} C_VEL
LIN {X 0,Y 143.613,Z 768.224,A -85,B 0,C 180,E1 7913.606,E2 7913.606} C_VEL
LIN {X 0,Y 144.756,Z 772.464,A -85,B 0,C 180,E1 7905.603,E2 7905.603} C_VEL
LIN {X 0,Y 151.763,Z 777.767,A -85,B 0,C 180,E1 7895.063,E2 7895.063} C_VEL
LIN {X 0,Y 165.778,Z 782.167,A -85,B 0,C 180,E1 7885.464,E2 7885.464} C_VEL
LIN {X 0,Y 170.847,Z 783.304,A -85,B 0,C 180,E1 7883.021,E2 7883.021} C_VEL
LIN {X 0,Y 160.479,Z 794.545,A -85,B 0,C 180,E1 7877.324,E2 7877.324} C_VEL
LIN {X 0,Y 151.161,Z 804.514,A -85,B 0,C 180,E1 7870.408,E2 7870.408} C_VEL
LIN {X 0,Y 144.073,Z 812.491,A -85,B 0,C 180,E1 7862.773,E2 7862.773} C_VEL
LIN {X 0,Y 139.251,Z 818.784,A -85,B 0,C 180,E1 7854.235,E2 7854.235} C_VEL
LIN {X 0,Y 137.009,Z 823.146,A -85,B 0,C 180,E1 7845.575,E2 7845.575} C_VEL
LIN {X 0,Y 136.74,Z 825.658,A -85,B 0,C 180,E1 7837.563,E2 7837.563} C_VEL
LIN {X 0,Y 137.028,Z 826.604,A -85,B 0,C 180,E1 7831.557,E2 7831.557} C_VEL
LIN {X 0,Y 136.915,Z 826.625,A -85,B 0,C 180,E1 7826.231,E2 7826.231} C_VEL
LIN {X 0,Y 136.64,Z 825.722,A -85,B 0,C 180,E1 7819.459,E2 7819.459} C_VEL
LIN {X 0,Y 137.623,Z 823.076,A -85,B 0,C 180,E1 7810.813,E2 7810.813} C_VEL
LIN {X 0,Y 141.219,Z 818.434,A -85,B 0,C 180,E1 7801.681,E2 7801.681} C_VEL
LIN {X 0,Y 147.425,Z 812.123,A -85,B 0,C 180,E1 7793.356,E2 7793.356} C_VEL
LIN {X 0,Y 156.234,Z 803.805,A -85,B 0,C 180,E1 7785.767,E2 7785.767} C_VEL
LIN {X 0,Y 166.772,Z 793.896,A -85,B 0,C 180,E1 7779.339,E2 7779.339} C_VEL
LIN {X 0,Y 178.435,Z 782.436,A -85,B 0,C 180,E1 7773.97,E2 7773.97} C_VEL
LIN {X 0,Y 183.589,Z 776.969,A -85,B 0,C 180,E1 7771.888,E2 7771.888} C_VEL
LIN {X 0,Y 170.947,Z 778.169,A -85,B 0,C 180,E1 7767.519,E2 7767.519} C_VEL
LIN {X 0,Y 158.732,Z 778.416,A -85,B 0,C 180,E1 7761.04,E2 7761.04} C_VEL
LIN {X 0,Y 150.367,Z 777.652,A -85,B 0,C 180,E1 7753.457,E2 7753.457} C_VEL
LIN {X 0,Y 146.026,Z 776.484,A -85,B 0,C 180,E1 7745.894,E2 7745.894} C_VEL
LIN {X 0,Y 144.961,Z 775.145,A -85,B 0,C 180,E1 7739.179,E2 7739.179} C_VEL
LIN {X 0,Y 145.779,Z 773.928,A -85,B 0,C 180,E1 7733.698,E2 7733.698} C_VEL
LIN {X 0,Y 150.698,Z 771.61,A -85,B 0,C 180,E1 7724.608,E2 7724.608} C_VEL
LIN {X 0,Y 160.466,Z 768.513,A -85,B 0,C 180,E1 7716.107,E2 7716.107} C_VEL
LIN {X 0,Y 172.565,Z 765.153,A -85,B 0,C 180,E1 7709.728,E2 7709.728} C_VEL
LIN {X 0,Y 185.122,Z 761.606,A -85,B 0,C 180,E1 7705.182,E2 7705.182} C_VEL
LIN {X 0,Y 173.84,Z 772.23,A -85,B 0,C 180,E1 7700.419,E2 7700.419} C_VEL
LIN {X 0,Y 162.77,Z 781.817,A -85,B 0,C 180,E1 7694.45,E2 7694.45} C_VEL
LIN {X 0,Y 153.507,Z 789.357,A -85,B 0,C 180,E1 7687.754,E2 7687.754} C_VEL
LIN {X 0,Y 146.296,Z 795.04,A -85,B 0,C 180,E1 7680.382,E2 7680.382} C_VEL
LIN {X 0,Y 141.076,Z 799.169,A -85,B 0,C 180,E1 7672.064,E2 7672.064} C_VEL
LIN {X 0,Y 138.311,Z 801.42,A -85,B 0,C 180,E1 7663.802,E2 7663.802} C_VEL
LIN {X 0,Y 137.297,Z 802.117,A -85,B 0,C 180,E1 7655.852,E2 7655.852} C_VEL
LIN {X 0,Y 137.365,Z 801.543,A -85,B 0,C 180,E1 7648.332,E2 7648.332} C_VEL
LIN {X 0,Y 138.546,Z 799.66,A -85,B 0,C 180,E1 7640.446,E2 7640.446} C_VEL
LIN {X 0,Y 141.724,Z 795.964,A -85,B 0,C 180,E1 7631.916,E2 7631.916} C_VEL
LIN {X 0,Y 146.881,Z 790.756,A -85,B 0,C 180,E1 7624.172,E2 7624.172} C_VEL
LIN {X 0,Y 154.107,Z 783.792,A -85,B 0,C 180,E1 7616.975,E2 7616.975} C_VEL
LIN {X 0,Y 163.27,Z 774.921,A -85,B 0,C 180,E1 7610.439,E2 7610.439} C_VEL
LIN {X 0,Y 173.541,Z 764.413,A -85,B 0,C 180,E1 7604.873,E2 7604.873} C_VEL
LIN {X 0,Y 183.852,Z 753.098,A -85,B 0,C 180,E1 7600.414,E2 7600.414} C_VEL
LIN {X 0,Y 194.393,Z 740.483,A -85,B 0,C 180,E1 7596.631,E2 7596.631} C_VEL
LIN {X 0,Y 204.668,Z 726.757,A -85,B 0,C 180,E1 7593.424,E2 7593.424} C_VEL
LIN {X 0,Y 193.688,Z 733.398,A -85,B 0,C 180,E1 7591.026,E2 7591.026} C_VEL
LIN {X 0,Y 179.588,Z 741.399,A -85,B 0,C 180,E1 7586.807,E2 7586.807} C_VEL
LIN {X 0,Y 168.584,Z 747.448,A -85,B 0,C 180,E1 7582.309,E2 7582.309} C_VEL
LIN {X 0,Y 159.938,Z 752.457,A -85,B 0,C 180,E1 7577.463,E2 7577.463} C_VEL
LIN {X 0,Y 157.57,Z 753.878,A -85,B 0,C 180,E1 7575.822,E2 7575.822} C_VEL
LIN {X 0,Y 153.004,Z 757.034,A -85,B 0,C 180,E1 7573.254,E2 7573.254} C_VEL
LIN {X 0,Y 143.05,Z 764.442,A -85,B 0,C 180,E1 7567.73,E2 7567.73} C_VEL
LIN {X 0,Y 140.279,Z 766.739,A -85,B 0,C 180,E1 7564.976,E2 7564.976} C_VEL
LIN {X 0,Y 137.824,Z 769.902,A -85,B 0,C 180,E1 7559.17,E2 7559.17} C_VEL
LIN {X 0,Y 136.991,Z 772.815,A -85,B 0,C 180,E1 7553.295,E2 7553.295} C_VEL
LIN {X 0,Y 137.708,Z 776.392,A -85,B 0,C 180,E1 7546.138,E2 7546.138} C_VEL
LIN {X 0,Y 145.205,Z 781.892,A -85,B 0,C 180,E1 7534.292,E2 7534.292} C_VEL
LIN {X 0,Y 159.6,Z 786.205,A -85,B 0,C 180,E1 7524.366,E2 7524.366} C_VEL
LIN {X 0,Y 161.65,Z 786.706,A -85,B 0,C 180,E1 7523.3,E2 7523.3} C_VEL
LIN {X 0,Y 151.164,Z 797.354,A -85,B 0,C 180,E1 7517.24,E2 7517.24} C_VEL
LIN {X 0,Y 141.785,Z 806.736,A -85,B 0,C 180,E1 7509.768,E2 7509.768} C_VEL
LIN {X 0,Y 134.737,Z 814.281,A -85,B 0,C 180,E1 7501.296,E2 7501.296} C_VEL
LIN {X 0,Y 130.543,Z 819.741,A -85,B 0,C 180,E1 7492.517,E2 7492.517} C_VEL
LIN {X 0,Y 128.813,Z 823.469,A -85,B 0,C 180,E1 7483.466,E2 7483.466} C_VEL
LIN {X 0,Y 128.857,Z 825.376,A -85,B 0,C 180,E1 7475.789,E2 7475.789} C_VEL
LIN {X 0,Y 129.097,Z 825.948,A -85,B 0,C 180,E1 7470,E2 7470} C_VEL
LIN {X 0,Y 128.798,Z 825.762,A -85,B 0,C 180,E1 7463.76,E2 7463.76} C_VEL
LIN {X 0,Y 128.837,Z 824.274,A -85,B 0,C 180,E1 7455.62,E2 7455.62} C_VEL
LIN {X 0,Y 130.867,Z 821.091,A -85,B 0,C 180,E1 7446.464,E2 7446.464} C_VEL
LIN {X 0,Y 135.999,Z 815.74,A -85,B 0,C 180,E1 7436.94,E2 7436.94} C_VEL
LIN {X 0,Y 144.156,Z 808.453,A -85,B 0,C 180,E1 7428.252,E2 7428.252} C_VEL
LIN {X 0,Y 154.069,Z 799.85,A -85,B 0,C 180,E1 7421.165,E2 7421.165} C_VEL
LIN {X 0,Y 165.958,Z 789.15,A -85,B 0,C 180,E1 7414.977,E2 7414.977} C_VEL
LIN {X 0,Y 173.571,Z 781.962,A -85,B 0,C 180,E1 7411.808,E2 7411.808} C_VEL
LIN {X 0,Y 161.161,Z 782.65,A -85,B 0,C 180,E1 7406.928,E2 7406.928} C_VEL
LIN {X 0,Y 149.594,Z 782.501,A -85,B 0,C 180,E1 7399.929,E2 7399.929} C_VEL
LIN {X 0,Y 139.577,Z 780.858,A -85,B 0,C 180,E1 7387.407,E2 7387.407} C_VEL
LIN {X 0,Y 138.139,Z 779.193,A -85,B 0,C 180,E1 7378.754,E2 7378.754} C_VEL
LIN {X 0,Y 139.109,Z 777.97,A -85,B 0,C 180,E1 7372.98,E2 7372.98} C_VEL
LIN {X 0,Y 144.405,Z 775.652,A -85,B 0,C 180,E1 7363.506,E2 7363.506} C_VEL
LIN {X 0,Y 155.005,Z 772.536,A -85,B 0,C 180,E1 7354.566,E2 7354.566} C_VEL
LIN {X 0,Y 167.924,Z 769.173,A -85,B 0,C 180,E1 7347.998,E2 7347.998} C_VEL
LIN {X 0,Y 175.219,Z 767.289,A -85,B 0,C 180,E1 7345.258,E2 7345.258} C_VEL
LIN {X 0,Y 163.3,Z 777.502,A -85,B 0,C 180,E1 7339.939,E2 7339.939} C_VEL
LIN {X 0,Y 152.358,Z 786.131,A -85,B 0,C 180,E1 7333.557,E2 7333.557} C_VEL
LIN {X 0,Y 143.358,Z 792.815,A -85,B 0,C 180,E1 7326.359,E2 7326.359} C_VEL
LIN {X 0,Y 136.562,Z 797.712,A -85,B 0,C 180,E1 7318.419,E2 7318.419} C_VEL
LIN {X 0,Y 131.934,Z 801.061,A -85,B 0,C 180,E1 7309.479,E2 7309.479} C_VEL
LIN {X 0,Y 129.776,Z 802.618,A -85,B 0,C 180,E1 7300.656,E2 7300.656} C_VEL
LIN {X 0,Y 129.243,Z 802.719,A -85,B 0,C 180,E1 7292.661,E2 7292.661} C_VEL
LIN {X 0,Y 129.758,Z 801.656,A -85,B 0,C 180,E1 7284.695,E2 7284.695} C_VEL
LIN {X 0,Y 131.882,Z 799.057,A -85,B 0,C 180,E1 7275.96,E2 7275.96} C_VEL
LIN {X 0,Y 136.379,Z 794.622,A -85,B 0,C 180,E1 7267.135,E2 7267.135} C_VEL
LIN {X 0,Y 142.943,Z 788.675,A -85,B 0,C 180,E1 7259.295,E2 7259.295} C_VEL
LIN {X 0,Y 151.611,Z 780.914,A -85,B 0,C 180,E1 7252.169,E2 7252.169} C_VEL
LIN {X 0,Y 161.569,Z 771.669,A -85,B 0,C 180,E1 7246.123,E2 7246.123} C_VEL
LIN {X 0,Y 172.879,Z 760.418,A -85,B 0,C 180,E1 7240.811,E2 7240.811} C_VEL
LIN {X 0,Y 184.178,Z 748.093,A -85,B 0,C 180,E1 7236.538,E2 7236.538} C_VEL
LIN {X 0,Y 193.755,Z 736.598,A -85,B 0,C 180,E1 7233.429,E2 7233.429} C_VEL
LIN {X 0,Y 175.865,Z 746.053,A -85,B 0,C 180,E1 7228.528,E2 7228.528} C_VEL
LIN {X 0,Y 164.114,Z 752.059,A -85,B 0,C 180,E1 7223.953,E2 7223.953} C_VEL
LIN {X 0,Y 154.672,Z 757.102,A -85,B 0,C 180,E1 7218.859,E2 7218.859} C_VEL
LIN {X 0,Y 147.73,Z 761.143,A -85,B 0,C 180,E1 7213.704,E2 7213.704} C_VEL
